KUKA KRL program: MyProgram_061().src

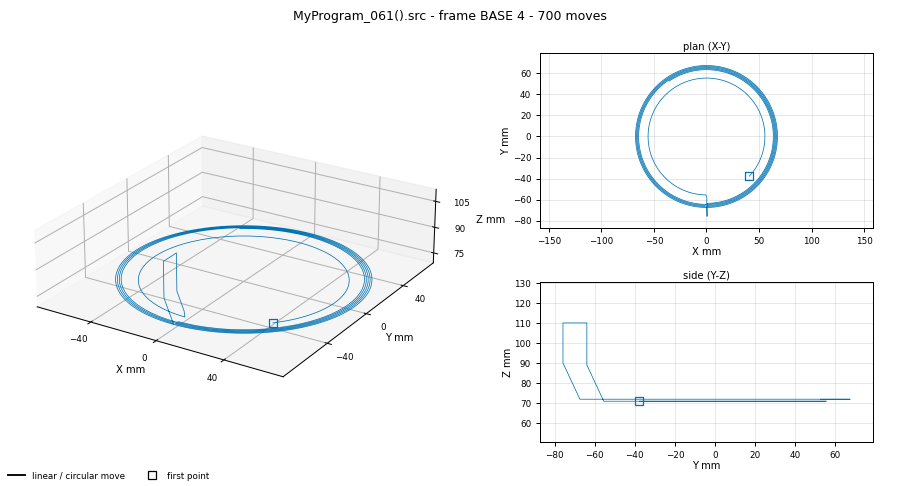
[picture p0: tool path of MyProgram_061().src in frame BASE 4, 700 of 700 moves have a stored position in this frame; points joined in program order, loops and branches not executed]
&ACCESS RVP
&REL 1
&PARAM TEMPLATE = C:\KRC\Roboter\Template\vorgabe
&PARAM EDITMASK = *
DEF MyProgram_061()
; ---- Setting reference (Base) ----
$BASE = BASE_DATA[4]

; --------------------------
; ---- Setting tool (TCP) ----
$TOOL = TOOL_DATA[3]
; --------------------------

$VEL.CP = VEL_APROX_PRINT
Startdeposition()
$VEL.CP = VEL_PRINT
LIN {X 40.7855,Y -37.7306,Z 71,A -48.0847,B 24.8792,C -2.5364,E1 25.1188,E2 491.8257} C_DIS
LIN {X 42.5102,Y -35.7771,Z 71,A -45.3429,B 24.8785,C -2.5444,E1 25.1238,E2 489.0774} C_DIS
LIN {X 44.2041,Y -33.6616,Z 71,A -42.6319,B 24.8779,C -2.5499,E1 25.1284,E2 486.3663} C_DIS
LIN {X 45.8213,Y -31.4249,Z 71,A -39.8032,B 24.8772,C -2.5572,E1 25.133,E2 483.534} C_DIS
LIN {X 47.3036,Y -29.1458,Z 71,A -37.0157,B 24.8765,C -2.5647,E1 25.1372,E2 480.7429} C_DIS
LIN {X 48.6728,Y -26.7969,Z 71,A -34.2291,B 24.8758,C -2.5723,E1 25.141,E2 477.9528} C_DIS
LIN {X 49.9338,Y -24.3666,Z 71,A -31.4273,B 24.875,C -2.58,E1 25.1445,E2 475.1476} C_DIS
LIN {X 51.0618,Y -21.9043,Z 71,A -28.6512,B 24.8743,C -2.588,E1 25.1477,E2 472.3679} C_DIS
LIN {X 52.067,Y -19.3938,Z 71,A -25.8775,B 24.8735,C -2.5961,E1 25.1505,E2 469.5904} C_DIS
LIN {X 52.9977,Y -16.6824,Z 71,A -22.8688,B 24.8725,C -2.6063,E1 25.1531,E2 466.5745} C_DIS
LIN {X 53.7819,Y -13.9471,Z 71,A -20.1757,B 24.8721,C -2.61,E1 25.1551,E2 463.8883} C_DIS
LIN {X 54.3576,Y -11.5051,Z 71,A -17.4095,B 24.8709,C -2.6221,E1 25.1568,E2 461.1095} C_DIS
LIN {X 54.8557,Y -8.8296,Z 71,A -14.6731,B 24.8702,C -2.6293,E1 25.1581,E2 458.372} C_DIS
LIN {X 55.2222,Y -6.1331,Z 71,A -11.877,B 24.8693,C -2.638,E1 25.159,E2 455.572} C_DIS
LIN {X 55.4575,Y -3.4024,Z 71,A -9.0827,B 24.8685,C -2.6462,E1 25.1596,E2 452.7749} C_DIS
LIN {X 55.5576,Y -0.6863,Z 71,A -6.4218,B 24.868,C -2.6518,E1 25.1598,E2 450.1164} C_DIS
LIN {X 55.5389,Y 1.5638,Z 71,A -3.9956,B 24.867,C -2.6615,E1 25.1596,E2 447.6817} C_DIS
LIN {X 55.3961,Y 4.2773,Z 71,A -1.3374,B 24.8664,C -2.6671,E1 25.1592,E2 445.0262} C_DIS
LIN {X 55.1439,Y 6.8016,Z 71,A 1.3866,B 24.8654,C -2.6776,E1 25.1583,E2 442.2934} C_DIS
LIN {X 54.7385,Y 9.5288,Z 71,A 4.1852,B 24.8646,C -2.6854,E1 25.1571,E2 439.4928} C_DIS
LIN {X 54.2118,Y 12.1736,Z 71,A 6.9784,B 24.8637,C -2.6941,E1 25.1555,E2 436.6953} C_DIS
LIN {X 53.5481,Y 14.8228,Z 71,A 9.7696,B 24.8629,C -2.702,E1 25.1535,E2 433.9015} C_DIS
LIN {X 52.7577,Y 17.428,Z 71,A 12.5599,B 24.8621,C -2.7099,E1 25.1511,E2 431.1084} C_DIS
LIN {X 51.8407,Y 19.9914,Z 71,A 15.3543,B 24.8613,C -2.7177,E1 25.1484,E2 428.3112} C_DIS
LIN {X 50.7941,Y 22.5183,Z 71,A 18.1681,B 24.8605,C -2.7255,E1 25.1453,E2 425.4943} C_DIS
LIN {X 49.6211,Y 24.997,Z 71,A 20.959,B 24.8598,C -2.7324,E1 25.1419,E2 422.7019} C_DIS
LIN {X 48.3402,Y 27.3922,Z 71,A 23.7438,B 24.859,C -2.7395,E1 25.1381,E2 419.9148} C_DIS
LIN {X 46.9433,Y 29.7227,Z 71,A 26.5321,B 24.8583,C -2.7464,E1 25.134,E2 417.1244} C_DIS
LIN {X 45.4343,Y 31.9818,Z 71,A 29.3209,B 24.8576,C -2.7531,E1 25.1296,E2 414.3334} C_DIS
LIN {X 43.7975,Y 34.1891,Z 71,A 32.1302,B 24.857,C -2.7593,E1 25.1248,E2 411.5228} C_DIS
LIN {X 42.0906,Y 36.2695,Z 71,A 34.9435,B 24.8562,C -2.7665,E1 25.1198,E2 408.7054} C_DIS
LIN {X 40.2294,Y 38.3236,Z 71,A 37.7223,B 24.8558,C -2.771,E1 25.1145,E2 405.9281} C_DIS
LIN {X 38.2353,Y 40.3127,Z 71,A 40.5586,B 24.8553,C -2.7755,E1 25.1088,E2 403.0929} C_DIS
LIN {X 36.2958,Y 42.0682,Z 71,A 43.3203,B 24.8546,C -2.7821,E1 25.103,E2 400.3266} C_DIS
LIN {X 34.1743,Y 43.809,Z 71,A 46.1312,B 24.8541,C -2.7868,E1 25.0969,E2 397.5151} C_DIS
LIN {X 32.0025,Y 45.4197,Z 71,A 48.9143,B 24.8536,C -2.7914,E1 25.0906,E2 394.7309} C_DIS
LIN {X 29.7582,Y 46.9206,Z 71,A 51.7458,B 24.8531,C -2.7967,E1 25.084,E2 391.8961} C_DIS
LIN {X 27.3868,Y 48.3433,Z 71,A 54.5334,B 24.8528,C -2.7994,E1 25.0773,E2 389.1106} C_DIS
LIN {X 24.9889,Y 49.6252,Z 71,A 57.3299,B 24.8524,C -2.8028,E1 25.0703,E2 386.3137} C_DIS
LIN {X 22.5309,Y 50.7884,Z 71,A 60.127,B 24.8521,C -2.8059,E1 25.0632,E2 383.5165} C_DIS
LIN {X 19.9947,Y 51.8394,Z 71,A 62.9475,B 24.8518,C -2.8085,E1 25.0559,E2 380.6962} C_DIS
LIN {X 17.4667,Y 52.7447,Z 71,A 65.7093,B 24.8516,C -2.8106,E1 25.0486,E2 377.9346} C_DIS
LIN {X 14.9277,Y 53.5184,Z 71,A 68.4748,B 24.8513,C -2.8131,E1 25.0412,E2 375.168} C_DIS
LIN {X 12.592,Y 54.1151,Z 71,A 70.7615,B 24.8516,C -2.8106,E1 25.035,E2 372.8907} C_DIS
LIN {X 10.1591,Y 54.6251,Z 71,A 73.4917,B 24.8511,C -2.8149,E1 25.0275,E2 370.1534} C_DIS
LIN {X 7.4737,Y 55.0568,Z 71,A 76.2953,B 24.8511,C -2.8156,E1 25.0198,E2 367.3507} C_DIS
LIN {X 4.7701,Y 55.3567,Z 71,A 79.1017,B 24.8511,C -2.816,E1 25.012,E2 364.5452} C_DIS
LIN {X 2.0552,Y 55.5237,Z 71,A 81.9069,B 24.8511,C -2.8159,E1 25.0042,E2 361.7412} C_DIS
LIN {X -0.664,Y 55.5577,Z 71,A 84.7191,B 24.8511,C -2.8155,E1 24.9963,E2 358.93} C_DIS
LIN {X -3.4053,Y 55.4574,Z 71,A 87.5443,B 24.8512,C -2.8144,E1 24.9884,E2 356.1067} C_DIS
LIN {X -6.1165,Y 55.2241,Z 71,A 90.3538,B 24.8513,C -2.8131,E1 24.9806,E2 353.2988} C_DIS
LIN {X -8.8133,Y 54.8583,Z 71,A 93.1693,B 24.8515,C -2.8114,E1 24.9729,E2 350.4849} C_DIS
LIN {X -11.5059,Y 54.3574,Z 71,A 96.0147,B 24.8517,C -2.8095,E1 24.9651,E2 347.6407} C_DIS
LIN {X -14.1791,Y 53.722,Z 71,A 98.8304,B 24.852,C -2.8065,E1 24.9575,E2 344.8282} C_DIS
LIN {X -16.7864,Y 52.9653,Z 71,A 101.6378,B 24.8524,C -2.8035,E1 24.95,E2 342.023} C_DIS
LIN {X -19.3546,Y 52.0818,Z 71,A 104.4495,B 24.8527,C -2.8003,E1 24.9426,E2 339.2136} C_DIS
LIN {X -21.8759,Y 51.074,Z 71,A 107.2582,B 24.8531,C -2.7965,E1 24.9353,E2 336.4075} C_DIS
LIN {X -24.3441,Y 49.9446,Z 71,A 110.0665,B 24.8535,C -2.7924,E1 24.9283,E2 333.6018} C_DIS
LIN {X -26.7824,Y 48.6807,Z 71,A 112.9149,B 24.854,C -2.788,E1 24.9212,E2 330.7559} C_DIS
LIN {X -29.1655,Y 47.2914,Z 71,A 115.7613,B 24.8545,C -2.783,E1 24.9144,E2 327.9129} C_DIS
LIN {X -31.4351,Y 45.8143,Z 71,A 118.5701,B 24.855,C -2.7779,E1 24.9079,E2 325.1068} C_DIS
LIN {X -33.7143,Y 44.1634,Z 71,A 121.4177,B 24.8558,C -2.7711,E1 24.9016,E2 322.2654} C_DIS
LIN {X -35.7726,Y 42.514,Z 71,A 124.2222,B 24.8562,C -2.7667,E1 24.8955,E2 319.4609} C_DIS
LIN {X -37.8107,Y 40.7119,Z 71,A 127.0522,B 24.8568,C -2.7607,E1 24.8897,E2 316.6336} C_DIS
LIN {X -39.8347,Y 38.7332,Z 71,A 129.9652,B 24.8576,C -2.7537,E1 24.8839,E2 313.725} C_DIS
LIN {X -41.6587,Y 36.7646,Z 71,A 132.8235,B 24.8581,C -2.7484,E1 24.8786,E2 310.8667} C_DIS
LIN {X -43.4432,Y 34.6373,Z 71,A 135.5659,B 24.8591,C -2.7391,E1 24.8737,E2 308.1339} C_DIS
LIN {X -45.0343,Y 32.5426,Z 71,A 138.3662,B 24.8597,C -2.7333,E1 24.8691,E2 305.3339} C_DIS
LIN {X -46.5685,Y 30.3066,Z 71,A 141.1834,B 24.8604,C -2.726,E1 24.8647,E2 302.52} C_DIS
LIN {X -47.9924,Y 27.997,Z 71,A 144.0124,B 24.8612,C -2.7187,E1 24.8607,E2 299.6939} C_DIS
LIN {X -49.3328,Y 25.561,Z 71,A 146.8831,B 24.862,C -2.7105,E1 24.8569,E2 296.8276} C_DIS
LIN {X -50.5224,Y 23.1212,Z 71,A 149.7025,B 24.8628,C -2.7026,E1 24.8535,E2 294.0117} C_DIS
LIN {X -51.5925,Y 20.6235,Z 71,A 152.525,B 24.8636,C -2.6946,E1 24.8505,E2 291.1927} C_DIS
LIN {X -52.5394,Y 18.0757,Z 71,A 155.3492,B 24.8645,C -2.6864,E1 24.8479,E2 288.372} C_DIS
LIN {X -53.3604,Y 15.4846,Z 71,A 158.172,B 24.8653,C -2.6782,E1 24.8456,E2 285.5528} C_DIS
LIN {X -54.0535,Y 12.8577,Z 71,A 160.9937,B 24.8662,C -2.6698,E1 24.8437,E2 282.7347} C_DIS
LIN {X -54.6257,Y 10.1558,Z 71,A 163.8614,B 24.867,C -2.6612,E1 24.8421,E2 279.8705} C_DIS
LIN {X -55.0575,Y 7.469,Z 71,A 166.6885,B 24.8679,C -2.6527,E1 24.841,E2 277.0469} C_DIS
LIN {X -55.3572,Y 4.7635,Z 71,A 169.5161,B 24.8687,C -2.6442,E1 24.8402,E2 274.2227} C_DIS
LIN {X -55.5241,Y 2.0464,Z 71,A 172.3494,B 24.8696,C -2.6357,E1 24.8398,E2 271.3926} C_DIS
LIN {X -55.56,Y -0.4299,Z 71,A 174.8514,B 24.8704,C -2.6269,E1 24.8398,E2 268.8967} C_DIS
LIN {X -55.4828,Y -2.9443,Z 71,A 177.5293,B 24.8711,C -2.6201,E1 24.8401,E2 266.2188} C_DIS
LIN {X -55.2942,Y -5.4464,Z 71,A -179.8635,B 24.8719,C -2.6123,E1 24.8408,E2 263.6146} C_DIS
LIN {X -54.9612,Y -8.1474,Z 71,A -177.0114,B 24.8727,C -2.6044,E1 24.8418,E2 260.7645} C_DIS
LIN {X -54.4945,Y -10.8382,Z 71,A -174.2087,B 24.8735,C -2.5955,E1 24.8433,E2 257.9663} C_DIS
LIN {X -53.9151,Y -13.425,Z 71,A -171.4694,B 24.8743,C -2.5874,E1 24.845,E2 255.2304} C_DIS
LIN {X -53.1514,Y -16.1868,Z 71,A -168.5076,B 24.8752,C -2.5787,E1 24.8473,E2 252.2722} C_DIS
LIN {X -52.3124,Y -18.7222,Z 71,A -165.7033,B 24.8759,C -2.5715,E1 24.8499,E2 249.4691} C_DIS
LIN {X -51.3364,Y -21.2529,Z 71,A -162.8859,B 24.8766,C -2.5639,E1 24.8528,E2 246.6542} C_DIS
LIN {X -50.2388,Y -23.731,Z 71,A -160.0738,B 24.8773,C -2.5565,E1 24.8561,E2 243.8446} C_DIS
LIN {X -49.0001,Y -26.1936,Z 71,A -157.2124,B 24.878,C -2.5491,E1 24.8597,E2 240.9854} C_DIS
LIN {X -47.6589,Y -28.5612,Z 71,A -154.3882,B 24.8787,C -2.5421,E1 24.8637,E2 238.1633} C_DIS
LIN {X -46.1931,Y -30.8757,Z 71,A -151.55,B 24.8794,C -2.5352,E1 24.868,E2 235.3274} C_DIS
LIN {X -44.6291,Y -33.0961,Z 71,A -148.7308,B 24.88,C -2.5287,E1 24.8726,E2 232.5099} C_DIS
LIN {X -42.9587,Y -35.2372,Z 71,A -145.9154,B 24.8806,C -2.5224,E1 24.8776,E2 229.6963} C_DIS
LIN {X -41.1159,Y -37.3705,Z 71,A -143.3335,B 24.8817,C -2.5104,E1 24.8823,E2 227.1315} C_DIS
LIN {X -39.7683,Y -38.8021,Z 71,A -140.955,B 24.8815,C -2.5122,E1 24.8869,E2 224.7385} C_DIS
LIN {X -37.8194,Y -40.7039,Z 71,A -138.1256,B 24.882,C -2.5069,E1 24.8926,E2 221.91} C_DIS
LIN {X -35.7707,Y -42.5156,Z 71,A -135.3035,B 24.8825,C -2.5016,E1 24.8986,E2 219.0895} C_DIS
LIN {X -33.6515,Y -44.2118,Z 71,A -132.4917,B 24.883,C -2.4969,E1 24.9048,E2 216.2787} C_DIS
LIN {X -31.4296,Y -45.818,Z 71,A -129.6545,B 24.8834,C -2.4924,E1 24.9113,E2 213.4423} C_DIS
LIN {X -29.1493,Y -47.3015,Z 71,A -126.8378,B 24.8838,C -2.4884,E1 24.9179,E2 210.6261} C_DIS
LIN {X -26.7993,Y -48.6714,Z 71,A -124.0239,B 24.8841,C -2.4848,E1 24.9248,E2 207.8127} C_DIS
LIN {X -24.3849,Y -49.9247,Z 71,A -121.2021,B 24.8844,C -2.4817,E1 24.9318,E2 204.9908} C_DIS
LIN {X -21.9003,Y -51.0636,Z 71,A -118.3881,B 24.8847,C -2.4786,E1 24.939,E2 202.1774} C_DIS
LIN {X -19.4007,Y -52.0644,Z 71,A -115.6085,B 24.8849,C -2.4761,E1 24.9462,E2 199.3979} C_DIS
LIN {X -16.8768,Y -52.9361,Z 71,A -112.8159,B 24.8851,C -2.4747,E1 24.9536,E2 196.6035} C_DIS
LIN {X -14.1541,Y -53.7287,Z 71,A -109.9102,B 24.8853,C -2.4725,E1 24.9614,E2 193.6984} C_DIS
LIN {X -11.4997,Y -54.3587,Z 71,A -107.1003,B 24.8853,C -2.4711,E1 24.9691,E2 190.8882} C_DIS
LIN {X -8.8264,Y -54.8562,Z 71,A -104.2941,B 24.8855,C -2.4703,E1 24.9768,E2 188.0813} C_DIS
LIN {X -6.0909,Y -55.2268,Z 71,A -101.4709,B 24.8855,C -2.4694,E1 24.9846,E2 185.2583} C_DIS
LIN {X -3.424,Y -55.4561,Z 71,A -98.6835,B 24.8855,C -2.4699,E1 24.9924,E2 182.4685} C_DIS
LIN {X -0.6806,Y -55.5576,Z 71,A -95.8539,B 24.8855,C -2.4703,E1 25.0003,E2 179.6376} C_DIS
LIN {X -0.6806,Y -55.5576,Z 71,A -95.8539,B 24.8855,C -2.4703,E1 25.0003,E2 179.6376} C_DIS
Enddeposition()
LIN {X 0.3163,Y -57.6707,Z 75.5315,A -95.798,B 24.8876,C -2.4468,E1 25.0003,E2 179.6376} C_DIS
LIN {X 0.3163,Y -64.01,Z 89.1262,A -95.7703,B 24.8887,C -2.4352,E1 25.0003,E2 179.6376} C_DIS
LIN {X 0.3163,Y -64.01,Z 110.1262,A -96.1254,B 24.8746,C -2.5845,E1 25.0003,E2 179.6376} C_DIS
LIN {X 0.541,Y -75.9406,Z 110.1262,A -95.0218,B 24.8919,C -2.4005,E1 25.0022,E2 178.9714} C_DIS
LIN {X 0.541,Y -75.9406,Z 90.1262,A -94.6838,B 24.9043,C -2.2582,E1 25.0022,E2 178.9714} C_DIS
LIN {X 0.4673,Y -69.6018,Z 76.5315,A -94.7092,B 24.9034,C -2.2689,E1 25.0022,E2 178.9714} C_DIS
LIN {X 0.4427,Y -67.4888,Z 72,A -94.7192,B 24.9031,C -2.2731,E1 25.0022,E2 178.9714} C_DIS
Startdeposition()
$VEL.CP = VEL_PRINT
LIN {X 3.0465,Y -67.4239,Z 72,A -92.1859,B 24.9023,C -2.2817,E1 25.0093,E2 176.4184} C_DIS
LIN {X 6.0645,Y -67.2198,Z 72,A -89.6068,B 24.9022,C -2.2832,E1 25.0165,E2 173.837} C_DIS
LIN {X 9.1586,Y -66.8693,Z 72,A -86.9568,B 24.902,C -2.285,E1 25.0238,E2 171.1848} C_DIS
LIN {X 12.2813,Y -66.3668,Z 72,A -84.2475,B 24.9018,C -2.2877,E1 25.0313,E2 168.4721} C_DIS
LIN {X 15.4225,Y -65.7074,Z 72,A -81.5243,B 24.9016,C -2.2901,E1 25.0387,E2 165.7467} C_DIS
LIN {X 18.5712,Y -64.8876,Z 72,A -78.7625,B 24.9014,C -2.293,E1 25.0462,E2 162.9825} C_DIS
LIN {X 21.7049,Y -63.9076,Z 72,A -76.0971,B 24.9014,C -2.2933,E1 25.0532,E2 160.3215} C_DIS
LIN {X 24.2902,Y -62.9701,Z 72,A -73.6943,B 24.9009,C -2.2981,E1 25.0595,E2 157.9123} C_DIS
LIN {X 27.1714,Y -61.7821,Z 72,A -71.1416,B 24.9008,C -2.2996,E1 25.0661,E2 155.3622} C_DIS
LIN {X 29.6034,Y -60.654,Z 72,A -68.807,B 24.9003,C -2.3047,E1 25.072,E2 153.0217} C_DIS
LIN {X 32.339,Y -59.2409,Z 72,A -66.2034,B 24.9,C -2.3088,E1 25.0784,E2 150.4157} C_DIS
LIN {X 34.9059,Y -57.7657,Z 72,A -63.7033,B 24.8996,C -2.313,E1 25.0844,E2 147.9133} C_DIS
LIN {X 37.4976,Y -56.1191,Z 72,A -61.0796,B 24.8991,C -2.3184,E1 25.0906,E2 145.2853} C_DIS
LIN {X 39.9919,Y -54.3685,Z 72,A -58.5313,B 24.8988,C -2.3227,E1 25.0964,E2 142.7359} C_DIS
LIN {X 42.3805,Y -52.5279,Z 72,A -55.9926,B 24.8983,C -2.3276,E1 25.1019,E2 140.195} C_DIS
LIN {X 44.7089,Y -50.562,Z 72,A -53.3854,B 24.8978,C -2.3339,E1 25.1074,E2 137.583} C_DIS
LIN {X 46.945,Y -48.4917,Z 72,A -50.8158,B 24.8973,C -2.3395,E1 25.1127,E2 135.0108} C_DIS
LIN {X 49.0787,Y -46.331,Z 72,A -48.2593,B 24.8968,C -2.3453,E1 25.1176,E2 132.4517} C_DIS
LIN {X 51.126,Y -44.063,Z 72,A -45.6236,B 24.8961,C -2.3529,E1 25.1225,E2 129.8098} C_DIS
LIN {X 53.0915,Y -41.6726,Z 72,A -43.0659,B 24.8957,C -2.3579,E1 25.127,E2 127.2522} C_DIS
LIN {X 54.915,Y -39.2379,Z 72,A -40.4951,B 24.8951,C -2.3646,E1 25.1312,E2 124.678} C_DIS
LIN {X 56.5978,Y -36.7707,Z 72,A -37.9346,B 24.8944,C -2.3722,E1 25.1352,E2 122.1121} C_DIS
LIN {X 58.206,Y -34.1668,Z 72,A -35.4034,B 24.8939,C -2.3778,E1 25.1388,E2 119.5808} C_DIS
LIN {X 59.6481,Y -31.5816,Z 72,A -32.9259,B 24.8933,C -2.3841,E1 25.1421,E2 117.1014} C_DIS
LIN {X 61.0128,Y -28.8569,Z 72,A -30.3627,B 24.8927,C -2.3911,E1 25.1453,E2 114.5355} C_DIS
LIN {X 62.1377,Y -26.3475,Z 72,A -27.976,B 24.892,C -2.3995,E1 25.1479,E2 112.1419} C_DIS
LIN {X 63.2638,Y -23.5158,Z 72,A -25.3796,B 24.8912,C -2.4076,E1 25.1505,E2 109.5408} C_DIS
LIN {X 64.2794,Y -20.5783,Z 72,A -22.9172,B 24.8909,C -2.4109,E1 25.1527,E2 107.0845} C_DIS
LIN {X 65.1078,Y -17.784,Z 72,A -20.3281,B 24.8899,C -2.4217,E1 25.1547,E2 104.4847} C_DIS
LIN {X 65.8872,Y -14.6361,Z 72,A -17.6072,B 24.8892,C -2.4295,E1 25.1564,E2 101.7613} C_DIS
LIN {X 66.5071,Y -11.4985,Z 72,A -14.9145,B 24.8885,C -2.4374,E1 25.1578,E2 99.0655} C_DIS
LIN {X 66.9708,Y -8.382,Z 72,A -12.2544,B 24.8878,C -2.4455,E1 25.1588,E2 96.402} C_DIS
LIN {X 67.2899,Y -5.2298,Z 72,A -9.6286,B 24.8871,C -2.4523,E1 25.1594,E2 93.7757} C_DIS
LIN {X 67.4554,Y -2.2519,Z 72,A -7.2372,B 24.8867,C -2.4565,E1 25.1597,E2 91.3886} C_DIS
LIN {X 67.4915,Y 0.4178,Z 72,A -4.8546,B 24.8858,C -2.4668,E1 25.1597,E2 88.9957} C_DIS
LIN {X 67.4063,Y 3.4277,Z 72,A -2.3161,B 24.8851,C -2.4744,E1 25.1595,E2 86.4544} C_DIS
LIN {X 67.1879,Y 6.4104,Z 72,A 0.2495,B 24.8843,C -2.4831,E1 25.1589,E2 83.8835} C_DIS
LIN {X 66.8007,Y 9.6406,Z 72,A 2.962,B 24.8836,C -2.4903,E1 25.1579,E2 81.1698} C_DIS
LIN {X 66.2999,Y 12.6333,Z 72,A 5.5603,B 24.8828,C -2.4989,E1 25.1566,E2 78.5667} C_DIS
LIN {X 65.6663,Y 15.5947,Z 72,A 8.0256,B 24.8823,C -2.5038,E1 25.1551,E2 76.1039} C_DIS
LIN {X 64.8876,Y 18.5712,Z 72,A 10.7132,B 24.8814,C -2.5137,E1 25.1531,E2 73.4084} C_DIS
LIN {X 63.9076,Y 21.7049,Z 72,A 13.4393,B 24.8808,C -2.5203,E1 25.1507,E2 70.6823} C_DIS
LIN {X 62.8914,Y 24.4943,Z 72,A 15.9577,B 24.8801,C -2.5275,E1 25.1482,E2 68.1608} C_DIS
LIN {X 61.7026,Y 27.3509,Z 72,A 18.5237,B 24.8795,C -2.5333,E1 25.1454,E2 65.5952} C_DIS
LIN {X 60.5094,Y 29.8978,Z 72,A 20.9549,B 24.8788,C -2.541,E1 25.1424,E2 63.1587} C_DIS
LIN {X 59.1291,Y 32.5443,Z 72,A 23.4386,B 24.8783,C -2.5465,E1 25.1392,E2 60.6751} C_DIS
LIN {X 57.6425,Y 35.1086,Z 72,A 25.9449,B 24.8777,C -2.5528,E1 25.1356,E2 58.1666} C_DIS
LIN {X 56.0135,Y 37.6538,Z 72,A 28.4811,B 24.8771,C -2.5586,E1 25.1317,E2 55.6296} C_DIS
LIN {X 54.1976,Y 40.2238,Z 72,A 31.1214,B 24.8766,C -2.5643,E1 25.1274,E2 52.9886} C_DIS
LIN {X 52.3853,Y 42.5564,Z 72,A 33.6271,B 24.876,C -2.5701,E1 25.123,E2 50.4808} C_DIS
LIN {X 50.4214,Y 44.8663,Z 72,A 36.1653,B 24.8755,C -2.575,E1 25.1184,E2 47.9425} C_DIS
LIN {X 48.339,Y 47.1035,Z 72,A 38.8042,B 24.8749,C -2.5817,E1 25.1133,E2 45.2991} C_DIS
LIN {X 46.1557,Y 49.2436,Z 72,A 41.3855,B 24.8744,C -2.5867,E1 25.1081,E2 42.7168} C_DIS
LIN {X 43.88,Y 51.2819,Z 72,A 43.9525,B 24.874,C -2.591,E1 25.1027,E2 40.1497} C_DIS
LIN {X 41.5192,Y 53.2126,Z 72,A 46.5487,B 24.8735,C -2.5958,E1 25.097,E2 37.5516} C_DIS
LIN {X 39.0793,Y 55.0281,Z 72,A 49.0988,B 24.8731,C -2.5994,E1 25.0912,E2 35.002} C_DIS
LIN {X 36.5704,Y 56.7265,Z 72,A 51.6334,B 24.8728,C -2.6025,E1 25.0853,E2 32.4685} C_DIS
LIN {X 33.9857,Y 58.3128,Z 72,A 54.2359,B 24.8724,C -2.607,E1 25.0791,E2 29.8635} C_DIS
LIN {X 31.4163,Y 59.7351,Z 72,A 56.6926,B 24.8722,C -2.6094,E1 25.0731,E2 27.4082} C_DIS
LIN {X 28.7113,Y 61.0818,Z 72,A 59.2802,B 24.8718,C -2.613,E1 25.0665,E2 24.8188} C_DIS
LIN {X 25.9706,Y 62.2965,Z 72,A 61.8519,B 24.8715,C -2.6164,E1 25.0599,E2 22.2451} C_DIS
LIN {X 23.2826,Y 63.3499,Z 72,A 64.2289,B 24.8715,C -2.6169,E1 25.0537,E2 19.8722} C_DIS
LIN {X 20.5783,Y 64.2794,Z 72,A 66.7005,B 24.8711,C -2.6199,E1 25.0472,E2 17.3981} C_DIS
LIN {X 17.7452,Y 65.1183,Z 72,A 69.2101,B 24.871,C -2.6216,E1 25.0404,E2 14.8886} C_DIS
LIN {X 14.6361,Y 65.8872,Z 72,A 71.9324,B 24.8708,C -2.6231,E1 25.033,E2 12.1665} C_DIS
LIN {X 11.4985,Y 66.5071,Z 72,A 74.6419,B 24.8708,C -2.624,E1 25.0256,E2 9.4579} C_DIS
LIN {X 8.382,Y 66.9708,Z 72,A 77.3195,B 24.8706,C -2.6247,E1 25.0182,E2 6.7809} C_DIS
LIN {X 5.2298,Y 67.2899,Z 72,A 79.9634,B 24.8707,C -2.6239,E1 25.0109,E2 4.1405} C_DIS
LIN {X 2.2519,Y 67.4554,Z 72,A 82.4866,B 24.8707,C -2.6236,E1 25.0038,E2 1.6189} C_DIS
LIN {X -0.7474,Y 67.4894,Z 72,A 85.0764,B 24.8707,C -2.6241,E1 24.9966,E2 -0.9719} C_DIS
LIN {X -3.8737,Y 67.3816,Z 72,A 87.6859,B 24.8709,C -2.6221,E1 24.9893,E2 -3.5774} C_DIS
LIN {X -6.8348,Y 67.146,Z 72,A 90.2461,B 24.8709,C -2.6218,E1 24.9822,E2 -6.1381} C_DIS
LIN {X -9.937,Y 66.7583,Z 72,A 92.9278,B 24.871,C -2.6208,E1 24.9748,E2 -8.8195} C_DIS
LIN {X -13.0653,Y 66.2168,Z 72,A 95.6433,B 24.8712,C -2.6192,E1 24.9673,E2 -11.534} C_DIS
LIN {X -16.2094,Y 65.5177,Z 72,A 98.3879,B 24.8714,C -2.6169,E1 24.9599,E2 -14.277} C_DIS
LIN {X -19.3582,Y 64.6572,Z 72,A 101.1678,B 24.8717,C -2.6142,E1 24.9524,E2 -17.0549} C_DIS
LIN {X -22.1483,Y 63.7555,Z 72,A 103.6299,B 24.872,C -2.6106,E1 24.9459,E2 -19.513} C_DIS
LIN {X -25.1936,Y 62.6149,Z 72,A 106.3976,B 24.8724,C -2.6071,E1 24.9387,E2 -22.2784} C_DIS
LIN {X -27.9427,Y 61.4372,Z 72,A 108.8432,B 24.873,C -2.6013,E1 24.9325,E2 -24.716} C_DIS
LIN {X -30.3456,Y 60.2863,Z 72,A 111.2055,B 24.873,C -2.6,E1 24.9266,E2 -27.0813} C_DIS
LIN {X -33.0501,Y 58.8471,Z 72,A 113.8218,B 24.8735,C -2.596,E1 24.9202,E2 -29.6954} C_DIS
LIN {X -35.6777,Y 57.292,Z 72,A 116.3871,B 24.874,C -2.5907,E1 24.914,E2 -32.2561} C_DIS
LIN {X -38.1834,Y 55.6547,Z 72,A 118.9897,B 24.8743,C -2.5871,E1 24.908,E2 -34.8589} C_DIS
LIN {X -40.6561,Y 53.8736,Z 72,A 121.5739,B 24.8749,C -2.5818,E1 24.9022,E2 -37.4396} C_DIS
LIN {X -43.0289,Y 51.998,Z 72,A 124.148,B 24.8754,C -2.5765,E1 24.8966,E2 -40.0106} C_DIS
LIN {X -45.3374,Y 49.9994,Z 72,A 126.8218,B 24.8758,C -2.5724,E1 24.891,E2 -42.6852} C_DIS
LIN {X -47.5542,Y 47.8946,Z 72,A 129.3811,B 24.8764,C -2.5656,E1 24.8859,E2 -45.2389} C_DIS
LIN {X -49.6741,Y 45.692,Z 72,A 131.9761,B 24.877,C -2.5592,E1 24.881,E2 -47.8301} C_DIS
LIN {X -51.691,Y 43.3985,Z 72,A 134.6032,B 24.8776,C -2.5534,E1 24.8762,E2 -50.4553} C_DIS
LIN {X -53.5973,Y 41.02,Z 72,A 137.2147,B 24.8782,C -2.5471,E1 24.8717,E2 -53.0642} C_DIS
LIN {X -55.4146,Y 38.529,Z 72,A 139.8081,B 24.8789,C -2.5396,E1 24.8675,E2 -55.6523} C_DIS
LIN {X -57.0869,Y 36.0061,Z 72,A 142.4013,B 24.8796,C -2.533,E1 24.8636,E2 -58.2428} C_DIS
LIN {X -58.6142,Y 33.4615,Z 72,A 144.947,B 24.8802,C -2.5264,E1 24.86,E2 -60.786} C_DIS
LIN {X -59.9534,Y 30.9994,Z 72,A 147.374,B 24.8807,C -2.5205,E1 24.8569,E2 -63.2117} C_DIS
LIN {X -61.2512,Y 28.3471,Z 72,A 149.751,B 24.8817,C -2.5105,E1 24.854,E2 -65.5776} C_DIS
LIN {X -62.3553,Y 25.8284,Z 72,A 152.1685,B 24.8822,C -2.5052,E1 24.8514,E2 -67.9959} C_DIS
LIN {X -63.3499,Y 23.2826,Z 72,A 154.5101,B 24.8828,C -2.4986,E1 24.8491,E2 -70.335} C_DIS
LIN {X -64.2794,Y 20.5783,Z 72,A 156.9047,B 24.8836,C -2.4905,E1 24.847,E2 -72.7239} C_DIS
LIN {X -65.1078,Y 17.784,Z 72,A 159.5197,B 24.884,C -2.4858,E1 24.845,E2 -75.3427} C_DIS
LIN {X -65.8872,Y 14.6361,Z 72,A 162.2791,B 24.8848,C -2.4773,E1 24.8432,E2 -78.098} C_DIS
LIN {X -66.5071,Y 11.4985,Z 72,A 165.0103,B 24.8856,C -2.4691,E1 24.8418,E2 -80.8258} C_DIS
LIN {X -66.9708,Y 8.382,Z 72,A 167.7085,B 24.8863,C -2.4611,E1 24.8408,E2 -83.521} C_DIS
LIN {X -67.2899,Y 5.2298,Z 72,A 170.3719,B 24.8872,C -2.4521,E1 24.8401,E2 -86.1788} C_DIS
LIN {X -67.4554,Y 2.2519,Z 72,A 172.9057,B 24.8879,C -2.4441,E1 24.8398,E2 -88.7088} C_DIS
LIN {X -67.4883,Y -0.8282,Z 72,A 175.6393,B 24.8884,C -2.4383,E1 24.8398,E2 -91.4449} C_DIS
LIN {X -67.3666,Y -4.1388,Z 72,A 178.4361,B 24.8893,C -2.4291,E1 24.8402,E2 -94.2367} C_DIS
LIN {X -67.1014,Y -7.2607,Z 72,A -178.9165,B 24.89,C -2.4205,E1 24.8409,E2 -96.8795} C_DIS
LIN {X -66.7041,Y -10.2871,Z 72,A -176.2767,B 24.8907,C -2.4135,E1 24.842,E2 -99.5183} C_DIS
LIN {X -66.1961,Y -13.1672,Z 72,A -173.8198,B 24.8914,C -2.4053,E1 24.8432,E2 -101.9702} C_DIS
LIN {X -65.5177,Y -16.2094,Z 72,A -171.0941,B 24.892,C -2.399,E1 24.845,E2 -104.6967} C_DIS
LIN {X -64.6572,Y -19.3582,Z 72,A -168.3022,B 24.8927,C -2.3912,E1 24.8471,E2 -107.4861} C_DIS
LIN {X -63.7555,Y -22.1483,Z 72,A -165.8304,B 24.8934,C -2.3835,E1 24.8493,E2 -109.9537} C_DIS
LIN {X -62.6149,Y -25.1936,Z 72,A -163.053,B 24.8941,C -2.3759,E1 24.8521,E2 -112.7286} C_DIS
LIN {X -61.4372,Y -27.9427,Z 72,A -160.5998,B 24.8949,C -2.367,E1 24.8549,E2 -115.174} C_DIS
LIN {X -60.2863,Y -30.3456,Z 72,A -158.2315,B 24.8952,C -2.3631,E1 24.8578,E2 -117.5457} C_DIS
LIN {X -58.8471,Y -33.0501,Z 72,A -155.6093,B 24.8958,C -2.3566,E1 24.8613,E2 -120.1662} C_DIS
LIN {X -57.292,Y -35.6777,Z 72,A -153.0395,B 24.8964,C -2.3494,E1 24.865,E2 -122.732} C_DIS
LIN {X -55.6547,Y -38.1834,Z 72,A -150.4334,B 24.8969,C -2.3444,E1 24.8691,E2 -125.3392} C_DIS
LIN {X -53.8736,Y -40.6561,Z 72,A -147.8471,B 24.8974,C -2.3382,E1 24.8734,E2 -127.9231} C_DIS
LIN {X -51.998,Y -43.0289,Z 72,A -145.272,B 24.8979,C -2.3324,E1 24.8779,E2 -130.4964} C_DIS
LIN {X -49.9994,Y -45.3374,Z 72,A -142.5983,B 24.8983,C -2.3284,E1 24.8829,E2 -133.1725} C_DIS
LIN {X -47.8946,Y -47.5542,Z 72,A -140.0405,B 24.8988,C -2.3221,E1 24.8878,E2 -135.7264} C_DIS
LIN {X -45.692,Y -49.6741,Z 72,A -137.448,B 24.8993,C -2.3168,E1 24.8931,E2 -138.3169} C_DIS
LIN {X -43.3985,Y -51.691,Z 72,A -134.8246,B 24.8997,C -2.3126,E1 24.8987,E2 -140.9404} C_DIS
LIN {X -41.02,Y -53.5973,Z 72,A -132.2312,B 24.9,C -2.3082,E1 24.9044,E2 -143.5328} C_DIS
LIN {X -38.529,Y -55.4146,Z 72,A -129.6413,B 24.9005,C -2.3032,E1 24.9103,E2 -146.1198} C_DIS
LIN {X -36.0061,Y -57.0869,Z 72,A -127.0448,B 24.9008,C -2.2999,E1 24.9163,E2 -148.7168} C_DIS
LIN {X -33.4615,Y -58.6142,Z 72,A -124.5074,B 24.901,C -2.2968,E1 24.9225,E2 -151.2544} C_DIS
LIN {X -30.8472,Y -60.0311,Z 72,A -121.994,B 24.9013,C -2.2933,E1 24.9287,E2 -153.7665} C_DIS
LIN {X -28.1059,Y -61.3621,Z 72,A -119.4231,B 24.9016,C -2.29,E1 24.9352,E2 -156.336} C_DIS
LIN {X -25.3076,Y -62.5685,Z 72,A -116.8629,B 24.9019,C -2.2867,E1 24.9417,E2 -158.8944} C_DIS
LIN {X -22.7376,Y -63.5472,Z 72,A -114.4786,B 24.9019,C -2.2858,E1 24.948,E2 -161.2813} C_DIS
LIN {X -19.7118,Y -64.5507,Z 72,A -111.6974,B 24.9019,C -2.2856,E1 24.9554,E2 -164.0669} C_DIS
LIN {X -16.5631,Y -65.4293,Z 72,A -108.9395,B 24.9022,C -2.2835,E1 24.9629,E2 -166.824} C_DIS
LIN {X -13.498,Y -66.1292,Z 72,A -106.4449,B 24.9026,C -2.2782,E1 24.9696,E2 -169.3091} C_DIS
LIN {X -10.717,Y -66.6377,Z 72,A -103.8593,B 24.9023,C -2.2819,E1 24.9768,E2 -171.9059} C_DIS
LIN {X -7.6073,Y -67.0631,Z 72,A -101.2066,B 24.9023,C -2.2811,E1 24.9841,E2 -174.5588} C_DIS
LIN {X -4.5313,Y -67.3404,Z 72,A -98.6084,B 24.9024,C -2.2805,E1 24.9914,E2 -177.1566} C_DIS
LIN {X -1.4981,Y -67.4766,Z 72,A -96.0673,B 24.9024,C -2.28,E1 24.9985,E2 -179.6968} C_DIS
LIN {X 0.4427,Y -67.4888,Z 72,A -94.7197,B 24.9031,C -2.2731,E1 25.0022,E2 -181.028} C_DIS
Enddeposition()
LIN {X 0.4427,Y -67.4888,Z 72,A -94.7197,B 24.9031,C -2.2731,E1 25.0022,E2 -181.028} C_DIS
Startdeposition()
$VEL.CP = VEL_PRINT
LIN {X -1.8903,Y -66.4875,Z 72,A -97.6111,B 24.9034,C -2.2687,E1 24.9941,E2 -178.1261} C_DIS
LIN {X -3.7975,Y -66.4058,Z 72,A -99.9353,B 24.9048,C -2.2529,E1 24.9875,E2 -175.7636} C_DIS
LIN {X -7.7565,Y -66.0604,Z 72,A -102.9874,B 24.904,C -2.2618,E1 24.9791,E2 -172.7307} C_DIS
LIN {X -11.7555,Y -65.4671,Z 72,A -106.308,B 24.9036,C -2.2665,E1 24.9699,E2 -169.4182} C_DIS
LIN {X -15.8202,Y -64.6054,Z 72,A -109.6264,B 24.903,C -2.2741,E1 24.9609,E2 -166.1137} C_DIS
LIN {X -18.6166,Y -63.8557,Z 72,A -112.2626,B 24.9031,C -2.2724,E1 24.9538,E2 -163.4694} C_DIS
LIN {X -21.2756,Y -63.0197,Z 72,A -114.7255,B 24.9031,C -2.2729,E1 24.9473,E2 -161.0031} C_DIS
LIN {X -24.2246,Y -61.9461,Z 72,A -117.4313,B 24.9029,C -2.2753,E1 24.9402,E2 -158.2973} C_DIS
LIN {X -27.0816,Y -60.7516,Z 72,A -119.9264,B 24.9023,C -2.2818,E1 24.9338,E2 -155.8122} C_DIS
LIN {X -30.7111,Y -58.9998,Z 72,A -123.5232,B 24.9022,C -2.2833,E1 24.9248,E2 -152.2093} C_DIS
LIN {X -32.6542,Y -57.9474,Z 72,A -125.5379,B 24.9022,C -2.2833,E1 24.9199,E2 -150.189} C_DIS
LIN {X -37.2856,Y -55.081,Z 72,A -129.9977,B 24.9011,C -2.2955,E1 24.9094,E2 -145.7437} C_DIS
LIN {X -39.5289,Y -53.4947,Z 72,A -132.5761,B 24.9011,C -2.2948,E1 24.9035,E2 -143.1549} C_DIS
LIN {X -41.9352,Y -51.6292,Z 72,A -135.2225,B 24.9008,C -2.2991,E1 24.8977,E2 -140.5087} C_DIS
LIN {X -43.9835,Y -49.8967,Z 72,A -137.5438,B 24.9005,C -2.3032,E1 24.8928,E2 -138.1883} C_DIS
LIN {X -46.2784,Y -47.7752,Z 72,A -140.2075,B 24.8999,C -2.3092,E1 24.8874,E2 -135.5279} C_DIS
LIN {X -48.3697,Y -45.6565,Z 72,A -142.7819,B 24.8995,C -2.3145,E1 24.8825,E2 -132.9549} C_DIS
LIN {X -50.3965,Y -43.4103,Z 72,A -145.4369,B 24.8991,C -2.3192,E1 24.8776,E2 -130.2994} C_DIS
LIN {X -52.0563,Y -41.4043,Z 72,A -147.7442,B 24.8987,C -2.3231,E1 24.8735,E2 -127.9905} C_DIS
LIN {X -53.4647,Y -39.5696,Z 72,A -149.7304,B 24.8983,C -2.328,E1 24.8702,E2 -126.0065} C_DIS
LIN {X -55.2907,Y -36.9759,Z 72,A -152.4302,B 24.8977,C -2.3355,E1 24.8659,E2 -123.3112} C_DIS
LIN {X -56.6684,Y -34.8269,Z 72,A -154.7142,B 24.8973,C -2.3394,E1 24.8625,E2 -121.0248} C_DIS
LIN {X -58.2658,Y -32.0833,Z 72,A -157.3909,B 24.8966,C -2.3478,E1 24.8589,E2 -118.3542} C_DIS
LIN {X -59.6257,Y -29.4773,Z 72,A -159.6069,B 24.8954,C -2.3611,E1 24.8561,E2 -116.1582} C_DIS
LIN {X -60.6778,Y -27.2461,Z 72,A -162.2325,B 24.8958,C -2.3569,E1 24.853,E2 -113.5081} C_DIS
LIN {X -62.2864,Y -23.3364,Z 72,A -165.8387,B 24.8948,C -2.368,E1 24.8493,E2 -109.9083} C_DIS
LIN {X -63.6264,Y -19.3876,Z 72,A -169.3816,B 24.8937,C -2.3795,E1 24.8462,E2 -106.3727} C_DIS
LIN {X -64.4748,Y -16.3456,Z 72,A -172.1163,B 24.893,C -2.3874,E1 24.8443,E2 -103.6409} C_DIS
LIN {X -65.2819,Y -12.745,Z 72,A -175.3901,B 24.8923,C -2.3952,E1 24.8424,E2 -100.3665} C_DIS
LIN {X -65.8217,Y -9.5741,Z 72,A -178.1276,B 24.8915,C -2.4044,E1 24.8412,E2 -97.6347} C_DIS
LIN {X -66.2133,Y -6.3226,Z 72,A 179.0603,B 24.8907,C -2.4134,E1 24.8403,E2 -94.8272} C_DIS
LIN {X -66.4237,Y -3.4727,Z 72,A 176.7966,B 24.8896,C -2.4251,E1 24.8399,E2 -92.5777} C_DIS
LIN {X -66.511,Y -0.7311,Z 72,A 174.172,B 24.8894,C -2.4273,E1 24.8398,E2 -89.9427} C_DIS
LIN {X -66.4712,Y 2.3989,Z 72,A 171.499,B 24.8886,C -2.4363,E1 24.84,E2 -87.2751} C_DIS
LIN {X -66.2997,Y 5.3376,Z 72,A 168.9504,B 24.8879,C -2.4441,E1 24.8405,E2 -84.7297} C_DIS
LIN {X -66.0058,Y 8.2117,Z 72,A 166.4414,B 24.8872,C -2.4516,E1 24.8412,E2 -82.2237} C_DIS
LIN {X -65.5841,Y 11.0848,Z 72,A 164.0005,B 24.8864,C -2.4607,E1 24.8423,E2 -79.7899} C_DIS
LIN {X -65.174,Y 13.2846,Z 72,A 161.9952,B 24.8859,C -2.4652,E1 24.8434,E2 -77.7836} C_DIS
LIN {X -64.461,Y 16.3995,Z 72,A 159.1586,B 24.8853,C -2.4721,E1 24.8452,E2 -74.9469} C_DIS
LIN {X -63.5907,Y 19.5037,Z 72,A 156.4405,B 24.8844,C -2.4819,E1 24.8474,E2 -72.2363} C_DIS
LIN {X -62.3809,Y 23.082,Z 72,A 153.1122,B 24.8836,C -2.4903,E1 24.8504,E2 -68.9093} C_DIS
LIN {X -61.2097,Y 26.0295,Z 72,A 150.3531,B 24.8829,C -2.498,E1 24.8534,E2 -66.1532} C_DIS
LIN {X -60.0078,Y 28.6918,Z 72,A 147.2526,B 24.8833,C -2.4938,E1 24.8571,E2 -63.026} C_DIS
LIN {X -57.8819,Y 32.7714,Z 72,A 143.8192,B 24.8812,C -2.5157,E1 24.8616,E2 -59.6266} C_DIS
LIN {X -56.2388,Y 35.5163,Z 72,A 141.0781,B 24.8804,C -2.5237,E1 24.8656,E2 -56.8906} C_DIS
LIN {X -54.5464,Y 38.0637,Z 72,A 138.7079,B 24.8793,C -2.5362,E1 24.8693,E2 -54.5386} C_DIS
LIN {X -53.4828,Y 39.5451,Z 72,A 136.8407,B 24.8794,C -2.5344,E1 24.8724,E2 -52.658} C_DIS
LIN {X -51.6671,Y 41.8885,Z 72,A 134.3135,B 24.8787,C -2.5416,E1 24.8768,E2 -50.1361} C_DIS
LIN {X -49.7184,Y 44.1844,Z 72,A 130.9266,B 24.8796,C -2.5321,E1 24.8831,E2 -46.7113} C_DIS
LIN {X -47.4328,Y 46.6292,Z 72,A 128.9479,B 24.8772,C -2.5574,E1 24.8868,E2 -44.7844} C_DIS
LIN {X -44.869,Y 49.1002,Z 72,A 125.5496,B 24.8772,C -2.5577,E1 24.8938,E2 -41.3728} C_DIS
LIN {X -41.9174,Y 51.6431,Z 72,A 121.8749,B 24.8772,C -2.5585,E1 24.9017,E2 -37.686} C_DIS
LIN {X -39.1013,Y 53.8078,Z 72,A 119.2755,B 24.8756,C -2.5742,E1 24.9074,E2 -35.1148} C_DIS
LIN {X -36.7655,Y 55.4298,Z 72,A 116.8045,B 24.8752,C -2.5785,E1 24.9131,E2 -32.6458} C_DIS
LIN {X -34.1636,Y 57.0708,Z 72,A 114.2829,B 24.8744,C -2.586,E1 24.9191,E2 -30.1343} C_DIS
LIN {X -31.8262,Y 58.4059,Z 72,A 111.8306,B 24.8744,C -2.5872,E1 24.9251,E2 -27.6776} C_DIS
LIN {X -29.1411,Y 59.7909,Z 72,A 109.5029,B 24.8734,C -2.5972,E1 24.9308,E2 -25.3676} C_DIS
LIN {X -26.6782,Y 60.9296,Z 72,A 106.8348,B 24.8737,C -2.5936,E1 24.9377,E2 -22.6843} C_DIS
LIN {X -23.7464,Y 62.131,Z 72,A 104.0833,B 24.8734,C -2.5968,E1 24.9448,E2 -19.9344} C_DIS
LIN {X -20.7856,Y 63.1832,Z 72,A 101.3533,B 24.8731,C -2.5995,E1 24.952,E2 -17.2058} C_DIS
LIN {X -18.7402,Y 63.8198,Z 72,A 98.9606,B 24.8741,C -2.5897,E1 24.9585,E2 -14.7856} C_DIS
LIN {X -14.3236,Y 64.9538,Z 72,A 95.6624,B 24.8724,C -2.607,E1 24.9674,E2 -11.5243} C_DIS
LIN {X -11.3101,Y 65.5464,Z 72,A 93.0852,B 24.872,C -2.6106,E1 24.9744,E2 -8.9528} C_DIS
LIN {X -7.6665,Y 66.0709,Z 72,A 90.1719,B 24.8713,C -2.6183,E1 24.9824,E2 -6.0557} C_DIS
LIN {X -4.2606,Y 66.3778,Z 72,A 86.3265,B 24.8731,C -2.5995,E1 24.9933,E2 -2.1638} C_DIS
LIN {X -0.9715,Y 66.5073,Z 72,A 82.9978,B 24.8741,C -2.5891,E1 25.0026,E2 1.1897} C_DIS
LIN {X 2.9774,Y 66.4476,Z 72,A 80.9969,B 24.871,C -2.6212,E1 25.008,E2 3.114} C_DIS
LIN {X 5.1495,Y 66.3147,Z 72,A 78.7397,B 24.8719,C -2.6123,E1 25.0143,E2 5.3912} C_DIS
LIN {X 8.131,Y 66.0156,Z 72,A 76.0927,B 24.8721,C -2.6104,E1 25.0217,E2 8.0409} C_DIS
LIN {X 11.1676,Y 65.5703,Z 72,A 73.4983,B 24.8721,C -2.6107,E1 25.0288,E2 10.632} C_DIS
LIN {X 13.9303,Y 65.0392,Z 72,A 70.9795,B 24.8724,C -2.6074,E1 25.0357,E2 13.1555} C_DIS
LIN {X 17.0502,Y 64.2921,Z 72,A 68.3043,B 24.8724,C -2.6079,E1 25.043,E2 15.8255} C_DIS
LIN {X 19.8523,Y 63.4826,Z 72,A 65.8243,B 24.8724,C -2.6069,E1 25.0496,E2 18.3037} C_DIS
LIN {X 22.6609,Y 62.5351,Z 72,A 63.2629,B 24.8726,C -2.6045,E1 25.0563,E2 20.8656} C_DIS
LIN {X 25.4852,Y 61.4383,Z 72,A 60.3696,B 24.8736,C -2.5951,E1 25.0639,E2 23.7746} C_DIS
LIN {X 28.9238,Y 59.8963,Z 72,A 57.4053,B 24.8733,C -2.5981,E1 25.0713,E2 26.7241} C_DIS
LIN {X 31.4553,Y 58.607,Z 72,A 54.0372,B 24.8757,C -2.5727,E1 25.0798,E2 30.1428} C_DIS
LIN {X 34.7572,Y 56.711,Z 72,A 51.6675,B 24.8741,C -2.59,E1 25.0853,E2 32.4643} C_DIS
LIN {X 37.2976,Y 55.0729,Z 72,A 49.0668,B 24.8745,C -2.5859,E1 25.0914,E2 35.0659} C_DIS
LIN {X 38.9885,Y 53.8897,Z 72,A 47.1602,B 24.8751,C -2.5798,E1 25.0957,E2 36.9805} C_DIS
LIN {X 41.331,Y 52.1142,Z 72,A 44.3076,B 24.8763,C -2.5673,E1 25.102,E2 39.852} C_DIS
LIN {X 45.4697,Y 48.5454,Z 72,A 40.0767,B 24.876,C -2.57,E1 25.1108,E2 44.0598} C_DIS
LIN {X 47.6735,Y 46.3839,Z 72,A 37.4194,B 24.8765,C -2.5644,E1 25.116,E2 46.7189} C_DIS
LIN {X 49.7688,Y 44.128,Z 72,A 34.4743,B 24.8778,C -2.5512,E1 25.1216,E2 49.6823} C_DIS
LIN {X 53.2549,Y 39.8505,Z 72,A 29.4479,B 24.8796,C -2.5331,E1 25.1302,E2 54.7278} C_DIS
LIN {X 55.8702,Y 36.0928,Z 72,A 26.1913,B 24.8788,C -2.5407,E1 25.1353,E2 57.9503} C_DIS
LIN {X 57.9279,Y 32.6892,Z 72,A 22.757,B 24.8797,C -2.5315,E1 25.1401,E2 61.3887} C_DIS
LIN {X 59.3338,Y 30.0603,Z 72,A 20.1959,B 24.8804,C -2.5247,E1 25.1434,E2 63.9523} C_DIS
LIN {X 60.7529,Y 27.0786,Z 72,A 17.4049,B 24.881,C -2.5181,E1 25.1467,E2 66.7436} C_DIS
LIN {X 61.6418,Y 24.9886,Z 72,A 15.3775,B 24.8817,C -2.5107,E1 25.1489,E2 68.7774} C_DIS
LIN {X 62.8224,Y 21.852,Z 72,A 12.54,B 24.8823,C -2.5036,E1 25.1516,E2 71.6159} C_DIS
LIN {X 63.7896,Y 18.842,Z 72,A 9.8774,B 24.883,C -2.4971,E1 25.1538,E2 74.2786} C_DIS
LIN {X 64.9318,Y 14.4244,Z 72,A 6.0409,B 24.8838,C -2.4877,E1 25.1563,E2 78.1152} C_DIS
LIN {X 65.7591,Y 9.995,Z 72,A 2.3633,B 24.8845,C -2.4811,E1 25.1581,E2 81.7868} C_DIS
LIN {X 66.3087,Y 5.225,Z 72,A -1.9665,B 24.8861,C -2.4631,E1 25.1594,E2 86.1336} C_DIS
LIN {X 66.5131,Y -0.3996,Z 72,A -6.4159,B 24.8866,C -2.4583,E1 25.1598,E2 90.5678} C_DIS
LIN {X 66.4457,Y -3.0147,Z 72,A -8.7614,B 24.8875,C -2.4488,E1 25.1596,E2 92.922} C_DIS
LIN {X 66.2995,Y -5.3395,Z 72,A -11.019,B 24.8887,C -2.4357,E1 25.1591,E2 95.1969} C_DIS
LIN {X 65.9905,Y -8.3327,Z 72,A -13.6308,B 24.8895,C -2.427,E1 25.1583,E2 97.8139} C_DIS
LIN {X 65.5232,Y -11.4418,Z 72,A -16.2926,B 24.8901,C -2.4197,E1 25.1571,E2 100.4774} C_DIS
LIN {X 65.1311,Y -13.4938,Z 72,A -18.2103,B 24.8909,C -2.4109,E1 25.156,E2 102.4047} C_DIS
LIN {X 64.5841,Y -15.9075,Z 72,A -20.1492,B 24.8911,C -2.4093,E1 25.1548,E2 104.3361} C_DIS
LIN {X 63.8286,Y -18.7095,Z 72,A -22.6327,B 24.8917,C -2.402,E1 25.1529,E2 106.8227} C_DIS
LIN {X 63.008,Y -21.3102,Z 72,A -24.9951,B 24.8924,C -2.3944,E1 25.1508,E2 109.1896} C_DIS
LIN {X 61.9174,Y -24.2975,Z 72,A -27.7719,B 24.8933,C -2.3851,E1 25.1481,E2 111.973} C_DIS
LIN {X 60.7099,Y -27.1749,Z 72,A -30.4435,B 24.8939,C -2.3775,E1 25.1451,E2 114.648} C_DIS
LIN {X 59.3256,Y -30.0764,Z 72,A -32.8222,B 24.8937,C -2.3796,E1 25.1422,E2 117.0088} C_DIS
LIN {X 58.2137,Y -32.177,Z 72,A -35.8618,B 24.8966,C -2.3478,E1 25.1381,E2 120.1078} C_DIS
LIN {X 56.0125,Y -35.8711,Z 72,A -38.8281,B 24.8958,C -2.3565,E1 25.1338,E2 123.0383} C_DIS
LIN {X 53.6295,Y -39.3448,Z 72,A -42.4782,B 24.8967,C -2.3461,E1 25.1279,E2 126.6952} C_DIS
LIN {X 51.7523,Y -41.7833,Z 72,A -45.1165,B 24.8973,C -2.3395,E1 25.1233,E2 129.3368} C_DIS
LIN {X 50.4799,Y -43.3125,Z 72,A -47.0555,B 24.8982,C -2.3293,E1 25.1198,E2 131.2911} C_DIS
LIN {X 47.7604,Y -46.2937,Z 72,A -50.2745,B 24.8984,C -2.3273,E1 25.1137,E2 134.5007} C_DIS
LIN {X 45.5489,Y -48.471,Z 72,A -52.9173,B 24.8989,C -2.3218,E1 25.1083,E2 137.1456} C_DIS
LIN {X 43.2816,Y -50.5061,Z 72,A -55.2331,B 24.8987,C -2.3237,E1 25.1035,E2 139.4475} C_DIS
LIN {X 41.5322,Y -51.9549,Z 72,A -57.8591,B 24.9005,C -2.3024,E1 25.0977,E2 142.114} C_DIS
LIN {X 38.3381,Y -54.3546,Z 72,A -60.9307,B 24.9003,C -2.3047,E1 25.0908,E2 145.1693} C_DIS
LIN {X 35.7619,Y -56.0826,Z 72,A -63.5771,B 24.9007,C -2.3003,E1 25.0847,E2 147.8176} C_DIS
LIN {X 32.8439,Y -57.8404,Z 72,A -67.3341,B 24.9029,C -2.2745,E1 25.0755,E2 151.6242} C_DIS
LIN {X 29.7151,Y -59.5079,Z 72,A -69.3766,B 24.9012,C -2.2946,E1 25.0705,E2 153.6136} C_DIS
LIN {X 27.2349,Y -60.6828,Z 72,A -71.9188,B 24.9019,C -2.2865,E1 25.064,E2 156.1684} C_DIS
LIN {X 24.8961,Y -61.6795,Z 72,A -74.1493,B 24.9023,C -2.2824,E1 25.0583,E2 158.4035} C_DIS
LIN {X 21.536,Y -62.9311,Z 72,A -77.1718,B 24.9025,C -2.2801,E1 25.0503,E2 161.4254} C_DIS
LIN {X 18.6187,Y -63.8551,Z 72,A -79.7924,B 24.9027,C -2.2775,E1 25.0433,E2 164.0475} C_DIS
LIN {X 15.5605,Y -64.6684,Z 72,A -82.1501,B 24.9022,C -2.2837,E1 25.037,E2 166.3869} C_DIS
LIN {X 12.916,Y -65.2486,Z 72,A -84.8184,B 24.903,C -2.2735,E1 25.0296,E2 169.076} C_DIS
LIN {X 8.4884,Y -65.9703,Z 72,A -88.6744,B 24.9032,C -2.271,E1 25.019,E2 172.9343} C_DIS
LIN {X 5.4517,Y -66.2905,Z 72,A -91.2534,B 24.9032,C -2.2708,E1 25.0118,E2 175.5121} C_DIS
LIN {X 2.4095,Y -66.4708,Z 72,A -93.9098,B 24.9034,C -2.269,E1 25.0044,E2 178.1718} C_DIS
LIN {X 0.4493,Y -66.5031,Z 72,A -95.7488,B 24.9037,C -2.2652,E1 24.9993,E2 180.0197} C_DIS
Enddeposition()
LIN {X 0.4493,Y -66.5031,Z 72,A -95.7488,B 24.9037,C -2.2652,E1 24.9993,E2 180.0197} C_DIS
Startdeposition()
$VEL.CP = VEL_PRINT
LIN {X 1.3322,Y -65.5222,Z 72,A -93.0585,B 24.8983,C -2.3276,E1 25.0072,E2 177.1816} C_DIS
LIN {X 6.4867,Y -65.2134,Z 72,A -89.0574,B 24.8992,C -2.3174,E1 25.0182,E2 173.2067} C_DIS
LIN {X 9.404,Y -64.8575,Z 72,A -86.6537,B 24.8994,C -2.3151,E1 25.0249,E2 170.8105} C_DIS
LIN {X 12.1699,Y -64.3959,Z 72,A -84.3808,B 24.8996,C -2.3127,E1 25.0311,E2 168.5458} C_DIS
LIN {X 16.6189,Y -63.3936,Z 72,A -80.1195,B 24.8987,C -2.3231,E1 25.0427,E2 164.2659} C_DIS
LIN {X 19.5765,Y -62.5435,Z 72,A -77.4453,B 24.8985,C -2.3258,E1 25.0499,E2 161.59} C_DIS
LIN {X 22.6629,Y -61.4924,Z 72,A -74.5397,B 24.8981,C -2.3308,E1 25.0575,E2 158.6785} C_DIS
LIN {X 25.7102,Y -60.282,Z 72,A -71.3425,B 24.897,C -2.3431,E1 25.0658,E2 155.4595} C_DIS
LIN {X 29.2046,Y -58.6687,Z 72,A -68.7956,B 24.8983,C -2.3279,E1 25.0722,E2 152.9552} C_DIS
LIN {X 33.1346,Y -56.5427,Z 72,A -64.9421,B 24.8979,C -2.3333,E1 25.0816,E2 149.1002} C_DIS
LIN {X 36.4297,Y -54.4787,Z 72,A -61.193,B 24.8965,C -2.3485,E1 25.0905,E2 145.3272} C_DIS
LIN {X 39.6195,Y -52.2031,Z 72,A -57.5311,B 24.8954,C -2.3616,E1 25.0988,E2 141.6474} C_DIS
LIN {X 42.2638,Y -50.0862,Z 72,A -54.7096,B 24.8951,C -2.3645,E1 25.1048,E2 138.8297} C_DIS
LIN {X 43.9423,Y -48.6217,Z 72,A -52.8171,B 24.8948,C -2.3675,E1 25.1088,E2 136.9377} C_DIS
LIN {X 46.1782,Y -46.503,Z 72,A -49.8435,B 24.8936,C -2.3811,E1 25.1148,E2 133.9442} C_DIS
LIN {X 48.6489,Y -43.9121,Z 72,A -46.8482,B 24.8932,C -2.3854,E1 25.1204,E2 130.9521} C_DIS
LIN {X 51.527,Y -40.4959,Z 72,A -43.2187,B 24.893,C -2.3883,E1 25.1268,E2 127.3325} C_DIS
LIN {X 53.297,Y -38.1361,Z 72,A -40.0696,B 24.891,C -2.4102,E1 25.132,E2 124.1468} C_DIS
LIN {X 55.1144,Y -35.4588,Z 72,A -36.7324,B 24.889,C -2.4315,E1 25.1371,E2 120.7759} C_DIS
LIN {X 57.2135,Y -31.9612,Z 72,A -34.3717,B 24.891,C -2.4098,E1 25.1403,E2 118.4788} C_DIS
LIN {X 58.7648,Y -29.0106,Z 72,A -31.5807,B 24.8905,C -2.415,E1 25.1439,E2 115.6902} C_DIS
LIN {X 59.779,Y -26.8587,Z 72,A -29.2508,B 24.8894,C -2.4278,E1 25.1466,E2 113.3428} C_DIS
LIN {X 60.9605,Y -24.0572,Z 72,A -25.9341,B 24.887,C -2.4533,E1 25.1501,E2 109.9841} C_DIS
LIN {X 62.0736,Y -21.0189,Z 72,A -23.9463,B 24.8883,C -2.4396,E1 25.1519,E2 108.0399} C_DIS
LIN {X 62.8363,Y -18.6148,Z 72,A -21.0234,B 24.8859,C -2.4655,E1 25.1542,E2 105.0724} C_DIS
LIN {X 63.9418,Y -14.3648,Z 72,A -17.2064,B 24.8848,C -2.4769,E1 25.1567,E2 101.2506} C_DIS
LIN {X 64.8101,Y -9.7289,Z 72,A -13.7227,B 24.8852,C -2.4729,E1 25.1583,E2 97.7969} C_DIS
LIN {X 65.1935,Y -6.6887,Z 72,A -11.0251,B 24.8844,C -2.4819,E1 25.1591,E2 95.094} C_DIS
LIN {X 65.5297,Y -0.9046,Z 72,A -5.7093,B 24.8823,C -2.5045,E1 25.1598,E2 89.7562} C_DIS
LIN {X 65.3845,Y 4.4481,Z 72,A -1.3667,B 24.8817,C -2.5103,E1 25.1593,E2 85.426} C_DIS
LIN {X 65.0272,Y 8.146,Z 72,A 1.9553,B 24.8806,C -2.5224,E1 25.1583,E2 82.095} C_DIS
LIN {X 64.5033,Y 11.5857,Z 72,A 5.0381,B 24.8796,C -2.5328,E1 25.1568,E2 79.0056} C_DIS
LIN {X 63.9727,Y 14.2291,Z 72,A 7.1709,B 24.8795,C -2.5341,E1 25.1556,E2 76.8822} C_DIS
LIN {X 63.0884,Y 17.7421,Z 72,A 10.0212,B 24.8793,C -2.5353,E1 25.1536,E2 74.0454} C_DIS
LIN {X 62.4069,Y 20.0082,Z 72,A 12.4185,B 24.8779,C -2.55,E1 25.1516,E2 71.627} C_DIS
LIN {X 61.185,Y 23.4798,Z 72,A 15.6609,B 24.877,C -2.56,E1 25.1485,E2 68.3792} C_DIS
LIN {X 59.778,Y 26.8611,Z 72,A 18.4502,B 24.8771,C -2.5583,E1 25.1454,E2 65.6092} C_DIS
LIN {X 58.7951,Y 28.9488,Z 72,A 20.8222,B 24.8757,C -2.5731,E1 25.1425,E2 63.2149} C_DIS
LIN {X 55.8629,Y 34.2684,Z 72,A 26.018,B 24.8746,C -2.5841,E1 25.1354,E2 58.02} C_DIS
LIN {X 54.0352,Y 37.0844,Z 72,A 29.4355,B 24.8727,C -2.6039,E1 25.13,E2 54.5725} C_DIS
LIN {X 51.2193,Y 40.8841,Z 72,A 32.8092,B 24.8736,C -2.5943,E1 25.1244,E2 51.2377} C_DIS
LIN {X 49.626,Y 42.8045,Z 72,A 35.1364,B 24.8728,C -2.603,E1 25.1201,E2 48.9005} C_DIS
LIN {X 48.0134,Y 44.6061,Z 72,A 37.3998,B 24.872,C -2.6114,E1 25.1159,E2 46.6272} C_DIS
LIN {X 45.8025,Y 46.8736,Z 72,A 40.525,B 24.8705,C -2.6262,E1 25.1096,E2 43.4801} C_DIS
LIN {X 42.8547,Y 49.5831,Z 72,A 43.6384,B 24.8708,C -2.6233,E1 25.1032,E2 40.386} C_DIS
LIN {X 40.1934,Y 51.7635,Z 72,A 46.5547,B 24.8705,C -2.6265,E1 25.0968,E2 37.4731} C_DIS
LIN {X 37.9798,Y 53.4085,Z 72,A 48.6554,B 24.8708,C -2.6229,E1 25.0921,E2 35.3883} C_DIS
LIN {X 36.2199,Y 54.6175,Z 72,A 50.9962,B 24.8694,C -2.6376,E1 25.0866,E2 33.0206} C_DIS
LIN {X 34.1932,Y 55.9086,Z 72,A 53.2089,B 24.8688,C -2.6435,E1 25.0814,E2 30.8009} C_DIS
LIN {X 31.1758,Y 57.6454,Z 72,A 56.128,B 24.8687,C -2.6446,E1 25.0742,E2 27.8878} C_DIS
LIN {X 27.5953,Y 59.4426,Z 72,A 59.3318,B 24.869,C -2.6415,E1 25.0662,E2 24.6997} C_DIS
LIN {X 24.2066,Y 60.9012,Z 72,A 62.7259,B 24.8682,C -2.6489,E1 25.0575,E2 21.296} C_DIS
LIN {X 22.2919,Y 61.6281,Z 72,A 64.5207,B 24.8681,C -2.6506,E1 25.0528,E2 19.5008} C_DIS
LIN {X 19.3206,Y 62.623,Z 72,A 67.2612,B 24.8679,C -2.6528,E1 25.0455,E2 16.7603} C_DIS
LIN {X 16.4003,Y 63.4504,Z 72,A 70.4998,B 24.8663,C -2.6683,E1 25.0367,E2 13.4899} C_DIS
LIN {X 11.7368,Y 64.4762,Z 72,A 73.6057,B 24.8686,C -2.645,E1 25.0283,E2 10.4432} C_DIS
LIN {X 9.6312,Y 64.825,Z 72,A 75.9254,B 24.8675,C -2.6561,E1 25.0219,E2 8.0994} C_DIS
LIN {X 6.7273,Y 65.1895,Z 72,A 78.5104,B 24.8675,C -2.6572,E1 25.0147,E2 5.5138} C_DIS
LIN {X 2.285,Y 65.496,Z 72,A 82.8477,B 24.8664,C -2.6673,E1 25.0025,E2 1.1539} C_DIS
LIN {X -1.7188,Y 65.5131,Z 72,A 86.1841,B 24.8669,C -2.6627,E1 24.9932,E2 -2.1718} C_DIS
LIN {X -6.3612,Y 65.226,Z 72,A 89.8289,B 24.868,C -2.6514,E1 24.9832,E2 -5.7912} C_DIS
LIN {X -8.8273,Y 64.9387,Z 72,A 92.1877,B 24.8677,C -2.6543,E1 24.9766,E2 -8.1586} C_DIS
LIN {X -11.3455,Y 64.5464,Z 72,A 94.2682,B 24.8682,C -2.6494,E1 24.9709,E2 -10.2294} C_DIS
LIN {X -14.2264,Y 63.9733,Z 72,A 96.9321,B 24.8682,C -2.6494,E1 24.9636,E2 -12.8964} C_DIS
LIN {X -19.4961,Y 62.5686,Z 72,A 101.2515,B 24.8697,C -2.6347,E1 24.9521,E2 -17.1875} C_DIS
LIN {X -21.9445,Y 61.7523,Z 72,A 103.9799,B 24.8689,C -2.6422,E1 24.9448,E2 -19.9389} C_DIS
LIN {X -24.8963,Y 60.6228,Z 72,A 107.6213,B 24.8674,C -2.6575,E1 24.9353,E2 -23.625} C_DIS
LIN {X -28.225,Y 59.1463,Z 72,A 109.9361,B 24.8697,C -2.6339,E1 24.9295,E2 -25.8893} C_DIS
LIN {X -30.3785,Y 58.0693,Z 72,A 111.9635,B 24.8702,C -2.6288,E1 24.9245,E2 -27.9101} C_DIS
LIN {X -32.8523,Y 56.7071,Z 72,A 114.5518,B 24.8704,C -2.6271,E1 24.9182,E2 -30.5019} C_DIS
LIN {X -35.5371,Y 55.0641,Z 72,A 117.2764,B 24.871,C -2.6214,E1 24.9118,E2 -33.2216} C_DIS
LIN {X -38.4185,Y 53.0944,Z 72,A 120.3382,B 24.8715,C -2.6156,E1 24.9048,E2 -36.28} C_DIS
LIN {X -41.4505,Y 50.7611,Z 72,A 123.7117,B 24.8722,C -2.6092,E1 24.8974,E2 -39.6506} C_DIS
LIN {X -43.997,Y 48.5717,Z 72,A 126.88,B 24.8724,C -2.6074,E1 24.8908,E2 -42.8272} C_DIS
LIN {X -46.3534,Y 46.3296,Z 72,A 129.4671,B 24.8735,C -2.5954,E1 24.8856,E2 -45.3966} C_DIS
LIN {X -48.7237,Y 43.8286,Z 72,A 132.5794,B 24.8741,C -2.5901,E1 24.8797,E2 -48.5098} C_DIS
LIN {X -50.7114,Y 41.513,Z 72,A 135.2339,B 24.8747,C -2.583,E1 24.875,E2 -51.1596} C_DIS
LIN {X -52.843,Y 38.7626,Z 72,A 138.4411,B 24.8752,C -2.5783,E1 24.8696,E2 -54.371} C_DIS
LIN {X -54.5845,Y 36.2698,Z 72,A 140.9848,B 24.8761,C -2.5687,E1 24.8656,E2 -56.9044} C_DIS
LIN {X -56.2216,Y 33.6771,Z 72,A 143.6665,B 24.8768,C -2.5613,E1 24.8617,E2 -59.582} C_DIS
LIN {X -58.1838,Y 30.1591,Z 72,A 147.0442,B 24.8781,C -2.5483,E1 24.8572,E2 -62.9465} C_DIS
LIN {X -59.1303,Y 28.2585,Z 72,A 149.2431,B 24.878,C -2.5497,E1 24.8545,E2 -65.1607} C_DIS
LIN {X -60.7632,Y 24.5515,Z 72,A 152.2687,B 24.88,C -2.5288,E1 24.8512,E2 -68.1532} C_DIS
LIN {X -62.2444,Y 20.5078,Z 72,A 156.3663,B 24.8804,C -2.5239,E1 24.8474,E2 -72.2623} C_DIS
LIN {X -63.0351,Y 17.9305,Z 72,A 158.7923,B 24.881,C -2.518,E1 24.8454,E2 -74.6882} C_DIS
LIN {X -63.8378,Y 14.8209,Z 72,A 161.5668,B 24.8819,C -2.5086,E1 24.8436,E2 -77.4564} C_DIS
LIN {X -64.448,Y 11.8939,Z 72,A 164.2162,B 24.8826,C -2.5011,E1 24.8421,E2 -80.1035} C_DIS
LIN {X -64.9964,Y 8.3893,Z 72,A 167.7289,B 24.8827,C -2.4995,E1 24.8408,E2 -83.6334} C_DIS
LIN {X -65.2983,Y 5.5805,Z 72,A 169.8947,B 24.884,C -2.4856,E1 24.8402,E2 -85.779} C_DIS
LIN {X -65.4801,Y 2.6993,Z 72,A 172.4728,B 24.8847,C -2.4787,E1 24.8398,E2 -88.3561} C_DIS
LIN {X -65.5341,Y -0.4698,Z 72,A 175.3356,B 24.8853,C -2.4718,E1 24.8398,E2 -91.2196} C_DIS
LIN {X -65.4343,Y -3.6423,Z 72,A 177.7317,B 24.8868,C -2.4555,E1 24.8401,E2 -93.5912} C_DIS
LIN {X -65.2696,Y -5.9006,Z 72,A -179.9763,B 24.8868,C -2.4555,E1 24.8406,E2 -95.8971} C_DIS
LIN {X -64.9178,Y -8.9806,Z 72,A -177.2633,B 24.8876,C -2.4472,E1 24.8416,E2 -98.6062} C_DIS
LIN {X -64.3165,Y -12.5833,Z 72,A -172.9618,B 24.8864,C -2.4598,E1 24.8438,E2 -102.9633} C_DIS
LIN {X -63.4022,Y -16.5861,Z 72,A -170.8421,B 24.8902,C -2.4192,E1 24.8452,E2 -104.9985} C_DIS
LIN {X -62.869,Y -18.5048,Z 72,A -167.8973,B 24.8884,C -2.4384,E1 24.8476,E2 -108.0061} C_DIS
LIN {X -61.834,Y -21.7129,Z 72,A -165.9457,B 24.891,C -2.4096,E1 24.8493,E2 -109.9} C_DIS
LIN {X -60.0602,Y -26.2239,Z 72,A -161.7324,B 24.8922,C -2.3969,E1 24.8537,E2 -114.1067} C_DIS
LIN {X -59.308,Y -27.8823,Z 72,A -160.0031,B 24.8923,C -2.3953,E1 24.8557,E2 -115.8415} C_DIS
LIN {X -58.095,Y -30.3294,Z 72,A -157.4659,B 24.8926,C -2.3918,E1 24.8589,E2 -118.3841} C_DIS
LIN {X -56.6203,Y -33.003,Z 72,A -154.3585,B 24.8925,C -2.3938,E1 24.8632,E2 -121.5123} C_DIS
LIN {X -54.9408,Y -35.7287,Z 72,A -151.9106,B 24.8938,C -2.3794,E1 24.8669,E2 -123.9382} C_DIS
LIN {X -52.718,Y -38.9333,Z 72,A -148.4569,B 24.8944,C -2.372,E1 24.8725,E2 -127.391} C_DIS
LIN {X -50.3089,Y -41.9994,Z 72,A -145.3374,B 24.8957,C -2.358,E1 24.8779,E2 -130.4919} C_DIS
LIN {X -48.6115,Y -43.9537,Z 72,A -142.7562,B 24.8955,C -2.3596,E1 24.8827,E2 -133.0885} C_DIS
LIN {X -46.4465,Y -46.2353,Z 72,A -140.0115,B 24.896,C -2.3537,E1 24.888,E2 -135.8309} C_DIS
LIN {X -43.574,Y -48.9515,Z 72,A -136.5767,B 24.8967,C -2.3464,E1 24.8951,E2 -139.2622} C_DIS
LIN {X -40.8252,Y -51.2667,Z 72,A -133.7734,B 24.8978,C -2.3334,E1 24.9011,E2 -142.0451} C_DIS
LIN {X -38.9695,Y -52.6915,Z 72,A -131.1485,B 24.8971,C -2.3423,E1 24.907,E2 -144.7007} C_DIS
LIN {X -36.6863,Y -54.3051,Z 72,A -128.7295,B 24.8974,C -2.3379,E1 24.9126,E2 -147.1173} C_DIS
LIN {X -33.8614,Y -56.1103,Z 72,A -125.9114,B 24.898,C -2.3311,E1 24.9192,E2 -149.928} C_DIS
LIN {X -30.7165,Y -57.8916,Z 72,A -123.1178,B 24.8991,C -2.3188,E1 24.926,E2 -152.7006} C_DIS
LIN {X -28.4391,Y -59.0435,Z 72,A -120.5996,B 24.8988,C -2.3225,E1 24.9324,E2 -155.2341} C_DIS
LIN {X -25.9793,Y -60.1668,Z 72,A -118.3469,B 24.8992,C -2.3175,E1 24.9381,E2 -157.4801} C_DIS
LIN {X -23.4721,Y -61.188,Z 72,A -115.8508,B 24.8992,C -2.3181,E1 24.9446,E2 -159.9832} C_DIS
LIN {X -20.6909,Y -62.1842,Z 72,A -113.2155,B 24.8992,C -2.3172,E1 24.9516,E2 -162.6213} C_DIS
LIN {X -16.6258,Y -63.3918,Z 72,A -109.4492,B 24.8994,C -2.3161,E1 24.9617,E2 -166.3911} C_DIS
LIN {X -12.9042,Y -64.2521,Z 72,A -106.2082,B 24.8997,C -2.3123,E1 24.9705,E2 -169.6272} C_DIS
LIN {X -9.7671,Y -64.8042,Z 72,A -103.2559,B 24.8994,C -2.3154,E1 24.9787,E2 -172.5895} C_DIS
LIN {X -6.9579,Y -65.1654,Z 72,A -101.1032,B 24.9001,C -2.3076,E1 24.9846,E2 -174.725} C_DIS
LIN {X -4.1496,Y -65.4045,Z 72,A -98.2324,B 24.8993,C -2.3171,E1 24.9927,E2 -177.6195} C_DIS
LIN {X -1.5016,Y -65.5187,Z 72,A -95.5795,B 24.8985,C -2.3254,E1 25.0001,E2 -180.2924} C_DIS
LIN {X -1.5016,Y -65.5187,Z 72,A -95.5795,B 24.8985,C -2.3254,E1 25.0001,E2 -180.2924} C_DIS
Enddeposition()
LIN {X 0.4521,Y -64.5472,Z 72,A -95.5516,B 24.9004,C -2.3035,E1 25.0001,E2 -180.2685} C_DIS
Startdeposition()
$VEL.CP = VEL_PRINT
LIN {X -2.0738,Y -64.5238,Z 72,A -97.697,B 24.9003,C -2.3052,E1 24.9941,E2 -178.1269} C_DIS
LIN {X -5.0206,Y -64.3616,Z 72,A -100.6303,B 24.9009,C -2.2981,E1 24.9858,E2 -175.1756} C_DIS
LIN {X -8.1995,Y -64.0343,Z 72,A -103.3885,B 24.9007,C -2.3002,E1 24.9782,E2 -172.4207} C_DIS
LIN {X -11.1268,Y -63.5914,Z 72,A -106.7071,B 24.902,C -2.2858,E1 24.969,E2 -169.0646} C_DIS
LIN {X -16.3378,Y -62.4557,Z 72,A -111.9027,B 24.9026,C -2.2784,E1 24.9548,E2 -163.8442} C_DIS
LIN {X -20.3353,Y -61.2712,Z 72,A -114.5511,B 24.9004,C -2.3037,E1 24.9479,E2 -161.2512} C_DIS
LIN {X -23.2733,Y -60.2159,Z 72,A -116.8093,B 24.8993,C -2.3172,E1 24.9421,E2 -159.0206} C_DIS
LIN {X -25.2276,Y -59.4234,Z 72,A -118.7514,B 24.8993,C -2.3175,E1 24.9371,E2 -157.0749} C_DIS
LIN {X -29.2485,Y -57.5511,Z 72,A -122.8363,B 24.8991,C -2.3189,E1 24.9267,E2 -152.9828} C_DIS
LIN {X -30.994,Y -56.63,Z 72,A -124.8574,B 24.8994,C -2.3154,E1 24.9217,E2 -150.9479} C_DIS
LIN {X -33.6019,Y -55.1229,Z 72,A -128.0513,B 24.9,C -2.3084,E1 24.914,E2 -147.7275} C_DIS
LIN {X -36.4971,Y -53.2514,Z 72,A -131.088,B 24.8996,C -2.3137,E1 24.907,E2 -144.6932} C_DIS
LIN {X -39.3491,Y -51.1788,Z 72,A -134.4007,B 24.8994,C -2.3154,E1 24.8996,E2 -141.3726} C_DIS
LIN {X -42.0988,Y -48.9429,Z 72,A -136.8857,B 24.8977,C -2.3347,E1 24.8944,E2 -138.924} C_DIS
LIN {X -45.6821,Y -45.6167,Z 72,A -141.3003,B 24.8971,C -2.3419,E1 24.8854,E2 -134.5084} C_DIS
LIN {X -47.864,Y -43.3216,Z 72,A -143.8756,B 24.8961,C -2.3527,E1 24.8806,E2 -131.9477} C_DIS
LIN {X -49.3638,Y -41.6043,Z 72,A -146.3923,B 24.8966,C -2.3474,E1 24.876,E2 -129.4068} C_DIS
LIN {X -51.9102,Y -38.3802,Z 72,A -150.5318,B 24.8966,C -2.3464,E1 24.869,E2 -125.2452} C_DIS
LIN {X -53.7779,Y -35.7155,Z 72,A -152.2334,B 24.894,C -2.377,E1 24.8664,E2 -123.6081} C_DIS
LIN {X -55.8859,Y -32.3173,Z 72,A -156.2425,B 24.894,C -2.377,E1 24.8605,E2 -119.5785} C_DIS
LIN {X -57.3081,Y -29.7228,Z 72,A -158.6077,B 24.8929,C -2.3892,E1 24.8574,E2 -117.2298} C_DIS
LIN {X -58.0789,Y -28.186,Z 72,A -160.4803,B 24.8931,C -2.3866,E1 24.8551,E2 -115.3409} C_DIS
LIN {X -59.3162,Y -25.48,Z 72,A -163.3075,B 24.8928,C -2.3904,E1 24.8519,E2 -112.5073} C_DIS
LIN {X -60.5681,Y -22.3413,Z 72,A -166.3484,B 24.8921,C -2.3982,E1 24.8489,E2 -109.4679} C_DIS
LIN {X -62.0392,Y -17.8536,Z 72,A -169.8395,B 24.8897,C -2.4241,E1 24.846,E2 -106.0186} C_DIS
LIN {X -62.7658,Y -15.1016,Z 72,A -173.4482,B 24.8909,C -2.411,E1 24.8435,E2 -102.3574} C_DIS
LIN {X -63.8413,Y -9.5905,Z 72,A -177.92,B 24.8886,C -2.436,E1 24.8413,E2 -97.9189} C_DIS
LIN {X -64.226,Y -6.5324,Z 72,A 179.3376,B 24.8879,C -2.4444,E1 24.8404,E2 -95.1801} C_DIS
LIN {X -64.4223,Y -4.1715,Z 72,A 176.9853,B 24.8877,C -2.4463,E1 24.84,E2 -92.8182} C_DIS
LIN {X -64.5557,Y 0.4377,Z 72,A 173.0812,B 24.8862,C -2.4627,E1 24.8398,E2 -88.93} C_DIS
LIN {X -64.4629,Y 3.4867,Z 72,A 170.4045,B 24.8853,C -2.4719,E1 24.8401,E2 -86.259} C_DIS
LIN {X -63.9886,Y 8.5486,Z 72,A 165.1242,B 24.8853,C -2.4717,E1 24.8418,E2 -80.9467} C_DIS
LIN {X -63.1882,Y 13.2262,Z 72,A 161.8616,B 24.8824,C -2.5029,E1 24.8434,E2 -77.7392} C_DIS
LIN {X -62.8126,Y 14.9061,Z 72,A 160.0286,B 24.8825,C -2.5018,E1 24.8446,E2 -75.893} C_DIS
LIN {X -61.9425,Y 18.1871,Z 72,A 156.7943,B 24.882,C -2.5069,E1 24.847,E2 -72.6522} C_DIS
LIN {X -60.7134,Y 21.9427,Z 72,A 153.1626,B 24.8812,C -2.5153,E1 24.8503,E2 -69.0197} C_DIS
LIN {X -58.949,Y 26.3169,Z 72,A 149.1006,B 24.8798,C -2.5302,E1 24.8547,E2 -64.9708} C_DIS
LIN {X -57.7035,Y 28.9472,Z 72,A 145.7692,B 24.8805,C -2.5235,E1 24.8589,E2 -61.6055} C_DIS
LIN {X -55.9893,Y 32.1374,Z 72,A 143.4201,B 24.878,C -2.5491,E1 24.8621,E2 -59.3054} C_DIS
LIN {X -54.4225,Y 34.7251,Z 72,A 140.8107,B 24.8772,C -2.5581,E1 24.8659,E2 -56.704} C_DIS
LIN {X -52.2032,Y 37.98,Z 72,A 136.8387,B 24.8772,C -2.5583,E1 24.8723,E2 -52.7131} C_DIS
LIN {X -49.8677,Y 40.9991,Z 72,A 133.7889,B 24.8756,C -2.5737,E1 24.8776,E2 -49.6855} C_DIS
LIN {X -47.7269,Y 43.472,Z 72,A 131.0764,B 24.8746,C -2.5846,E1 24.8826,E2 -46.9872} C_DIS
LIN {X -45.6688,Y 45.6302,Z 72,A 128.0043,B 24.8748,C -2.5826,E1 24.8886,E2 -43.897} C_DIS
LIN {X -43.1013,Y 48.0614,Z 72,A 125.076,B 24.8737,C -2.594,E1 24.8946,E2 -40.9839} C_DIS
LIN {X -40.9106,Y 49.9395,Z 72,A 122.3042,B 24.8735,C -2.5953,E1 24.9005,E2 -38.2048} C_DIS
LIN {X -37.7353,Y 52.3806,Z 72,A 118.3587,B 24.8735,C -2.5948,E1 24.9094,E2 -34.244} C_DIS
LIN {X -34.1011,Y 54.8156,Z 72,A 115.1278,B 24.8716,C -2.6152,E1 24.9169,E2 -31.0514} C_DIS
LIN {X -31.6903,Y 56.2441,Z 72,A 112.558,B 24.8713,C -2.6179,E1 24.9231,E2 -28.4802} C_DIS
LIN {X -30.0194,Y 57.1528,Z 72,A 110.5063,B 24.8718,C -2.6132,E1 24.9282,E2 -26.4118} C_DIS
LIN {X -26.4393,Y 58.8947,Z 72,A 107.1194,B 24.871,C -2.6216,E1 24.9368,E2 -23.0364} C_DIS
LIN {X -23.1025,Y 60.2817,Z 72,A 103.1948,B 24.872,C -2.6111,E1 24.9471,E2 -19.0784} C_DIS
LIN {X -19.7246,Y 61.4702,Z 72,A 100.9796,B 24.8696,C -2.6348,E1 24.9528,E2 -16.9155} C_DIS
LIN {X -15.3903,Y 62.6958,Z 72,A 96.8675,B 24.8695,C -2.6365,E1 24.9639,E2 -12.801} C_DIS
LIN {X -12.5129,Y 63.3334,Z 72,A 94.1468,B 24.8695,C -2.6365,E1 24.9713,E2 -10.077} C_DIS
LIN {X -10.021,Y 63.7745,Z 72,A 91.7168,B 24.8697,C -2.6341,E1 24.978,E2 -7.6391} C_DIS
LIN {X -6.7073,Y 64.2077,Z 72,A 89.2265,B 24.8685,C -2.646,E1 24.9849,E2 -5.1755} C_DIS
LIN {X -3.7934,Y 64.4459,Z 72,A 86.2754,B 24.8692,C -2.6393,E1 24.9931,E2 -2.2074} C_DIS
LIN {X 0.2217,Y 64.5569,Z 72,A 82.9863,B 24.8685,C -2.6462,E1 25.0023,E2 1.0655} C_DIS
LIN {X 5.3524,Y 64.3351,Z 72,A 78.275,B 24.8688,C -2.6429,E1 25.0154,E2 5.7828} C_DIS
LIN {X 8.4091,Y 64.007,Z 72,A 75.6303,B 24.8688,C -2.6443,E1 25.0227,E2 8.4222} C_DIS
LIN {X 10.8456,Y 63.6398,Z 72,A 73.0305,B 24.8697,C -2.6344,E1 25.03,E2 11.043} C_DIS
LIN {X 17.3515,Y 62.182,Z 72,A 67.4626,B 24.8692,C -2.6391,E1 25.045,E2 16.5918} C_DIS
LIN {X 20.3654,Y 61.2613,Z 72,A 64.1574,B 24.8706,C -2.6253,E1 25.0539,E2 19.9236} C_DIS
LIN {X 26.4918,Y 58.871,Z 72,A 58.8619,B 24.8699,C -2.6319,E1 25.0675,E2 25.1913} C_DIS
LIN {X 29.4885,Y 57.4286,Z 72,A 55.8902,B 24.8703,C -2.6278,E1 25.0749,E2 28.1647} C_DIS
LIN {X 31.9859,Y 56.076,Z 72,A 53.2759,B 24.8709,C -2.6221,E1 25.0813,E2 30.7846} C_DIS
LIN {X 35.921,Y 53.6414,Z 72,A 49.3886,B 24.871,C -2.6211,E1 25.0905,E2 34.6619} C_DIS
LIN {X 37.6999,Y 52.4056,Z 72,A 47.0768,B 24.8722,C -2.6086,E1 25.0958,E2 36.9953} C_DIS
LIN {X 42.029,Y 49.0023,Z 72,A 42.8891,B 24.8715,C -2.6165,E1 25.1048,E2 41.1484} C_DIS
LIN {X 44.9991,Y 46.2901,Z 72,A 38.9856,B 24.873,C -2.6012,E1 25.1128,E2 45.0722} C_DIS
LIN {X 46.9956,Y 44.2609,Z 72,A 36.5152,B 24.8734,C -2.5972,E1 25.1176,E2 47.5416} C_DIS
LIN {X 49.8423,Y 41.0299,Z 72,A 32.465,B 24.8747,C -2.5829,E1 25.125,E2 51.6071} C_DIS
LIN {X 53.0453,Y 36.7942,Z 72,A 27.5701,B 24.8763,C -2.567,E1 25.1331,E2 56.5161} C_DIS
LIN {X 55.0348,Y 33.7469,Z 72,A 24.1251,B 24.8776,C -2.5534,E1 25.1382,E2 59.9759} C_DIS
LIN {X 58.0362,Y 28.2743,Z 72,A 19.6061,B 24.8766,C -2.564,E1 25.144,E2 64.446} C_DIS
LIN {X 59.3029,Y 25.5102,Z 72,A 16.3322,B 24.8787,C -2.5419,E1 25.1478,E2 67.7543} C_DIS
LIN {X 60.5222,Y 22.4633,Z 72,A 13.4844,B 24.8794,C -2.5352,E1 25.1506,E2 70.6022} C_DIS
LIN {X 61.6421,Y 19.1801,Z 72,A 10.7854,B 24.8793,C -2.5357,E1 25.153,E2 73.2846} C_DIS
LIN {X 62.4011,Y 16.5423,Z 72,A 7.7651,B 24.8814,C -2.5136,E1 25.1552,E2 76.3398} C_DIS
LIN {X 63.2929,Y 12.7132,Z 72,A 4.8024,B 24.8811,C -2.5164,E1 25.157,E2 79.2787} C_DIS
LIN {X 63.745,Y 10.2117,Z 72,A 2.5307,B 24.8818,C -2.509,E1 25.158,E2 81.5546} C_DIS
LIN {X 64.1318,Y 7.398,Z 72,A -0.1623,B 24.883,C -2.4968,E1 25.159,E2 84.2606} C_DIS
LIN {X 64.4012,Y 4.4856,Z 72,A -2.3634,B 24.8828,C -2.4987,E1 25.1595,E2 86.444} C_DIS
LIN {X 64.5348,Y 1.6944,Z 72,A -5.3968,B 24.8849,C -2.4767,E1 25.1598,E2 89.5113} C_DIS
LIN {X 64.5495,Y -0.9985,Z 72,A -7.9571,B 24.886,C -2.4648,E1 25.1597,E2 92.0845} C_DIS
LIN {X 64.1913,Y -6.8635,Z 72,A -12.9881,B 24.8871,C -2.453,E1 25.1585,E2 97.1136} C_DIS
LIN {X 63.5853,Y -11.1611,Z 72,A -16.2805,B 24.8869,C -2.4552,E1 25.1571,E2 100.3815} C_DIS
LIN {X 63.1444,Y -13.431,Z 72,A -18.2923,B 24.8874,C -2.4497,E1 25.156,E2 102.3944} C_DIS
LIN {X 62.6758,Y -15.4724,Z 72,A -20.4988,B 24.8887,C -2.435,E1 25.1546,E2 104.6229} C_DIS
LIN {X 61.4921,Y -19.6563,Z 72,A -23.7088,B 24.8883,C -2.4397,E1 25.1521,E2 107.8034} C_DIS
LIN {X 60.0033,Y -23.8168,Z 72,A -28.083,B 24.8904,C -2.4162,E1 25.1478,E2 112.2089} C_DIS
LIN {X 58.744,Y -26.7729,Z 72,A -30.7116,B 24.8907,C -2.4133,E1 25.1449,E2 114.8298} C_DIS
LIN {X 57.1273,Y -30.0678,Z 72,A -34.2601,B 24.8922,C -2.3964,E1 25.1404,E2 118.3995} C_DIS
LIN {X 54.4299,Y -34.7135,Z 72,A -38.6635,B 24.8926,C -2.3921,E1 25.1342,E2 122.7903} C_DIS
LIN {X 52.7512,Y -37.2147,Z 72,A -41.5685,B 24.8938,C -2.379,E1 25.1295,E2 125.7122} C_DIS
LIN {X 51.1762,Y -39.3525,Z 72,A -44.2752,B 24.8951,C -2.3639,E1 25.1249,E2 128.4416} C_DIS
LIN {X 48.1795,Y -42.9694,Z 72,A -48.0346,B 24.8951,C -2.3635,E1 25.1181,E2 132.1848} C_DIS
LIN {X 44.5633,Y -46.7097,Z 72,A -53.0114,B 24.8969,C -2.3435,E1 25.1083,E2 137.1879} C_DIS
LIN {X 41.7357,Y -49.2521,Z 72,A -55.8141,B 24.8964,C -2.3501,E1 25.1024,E2 139.964} C_DIS
LIN {X 39.1372,Y -51.3411,Z 72,A -59.3051,B 24.8981,C -2.3307,E1 25.0947,E2 143.4879} C_DIS
LIN {X 36.133,Y -53.4979,Z 72,A -62.9283,B 24.8994,C -2.3159,E1 25.0863,E2 147.1338} C_DIS
LIN {X 33.3136,Y -55.2981,Z 72,A -64.9503,B 24.8978,C -2.3334,E1 25.0816,E2 149.1081} C_DIS
LIN {X 29.3365,Y -57.5064,Z 72,A -69.4626,B 24.8994,C -2.315,E1 25.0704,E2 153.651} C_DIS
LIN {X 25.1227,Y -59.4682,Z 72,A -73.2984,B 24.8994,C -2.3158,E1 25.0607,E2 157.4754} C_DIS
LIN {X 22.7172,Y -60.4282,Z 72,A -75.5903,B 24.8996,C -2.3128,E1 25.0547,E2 159.7693} C_DIS
LIN {X 19.7843,Y -61.4508,Z 72,A -78.3204,B 24.8999,C -2.3101,E1 25.0475,E2 162.5007} C_DIS
LIN {X 16.7333,Y -62.3508,Z 72,A -82.1628,B 24.9022,C -2.2833,E1 25.037,E2 166.4004} C_DIS
LIN {X 12.8423,Y -63.2668,Z 72,A -84.3249,B 24.8997,C -2.3124,E1 25.0313,E2 168.4907} C_DIS
LIN {X 9.9186,Y -63.7906,Z 72,A -87.3859,B 24.9007,C -2.3005,E1 25.0228,E2 171.5769} C_DIS
LIN {X 5.427,Y -64.3292,Z 72,A -91.0597,B 24.9002,C -2.306,E1 25.0126,E2 175.2349} C_DIS
LIN {X 3.5448,Y -64.4597,Z 72,A -93.3753,B 24.9016,C -2.2907,E1 25.006,E2 177.586} C_DIS
LIN {X 0.4521,Y -64.5472,Z 72,A -95.5504,B 24.9005,C -2.303,E1 25.0001,E2 179.7315} C_DIS
Enddeposition()
LIN {X 0.4521,Y -64.5472,Z 72,A -95.5504,B 24.9005,C -2.303,E1 25.0001,E2 179.7315} C_DIS
Startdeposition()
$VEL.CP = VEL_PRINT
LIN {X 0.8268,Y -63.5735,Z 72,A -93.9143,B 24.8964,C -2.3496,E1 25.0049,E2 177.9849} C_DIS
LIN {X 3.7418,Y -63.4688,Z 72,A -91.719,B 24.8972,C -2.3406,E1 25.011,E2 175.8117} C_DIS
LIN {X 6.5427,Y -63.241,Z 72,A -88.9358,B 24.8966,C -2.3478,E1 25.0188,E2 173.0133} C_DIS
LIN {X 9.1211,Y -62.921,Z 72,A -85.9334,B 24.8951,C -2.3648,E1 25.0272,E2 169.973} C_DIS
LIN {X 12.6945,Y -62.2983,Z 72,A -82.6394,B 24.8948,C -2.3682,E1 25.0362,E2 166.675} C_DIS
LIN {X 15.8352,Y -61.5749,Z 72,A -80.6581,B 24.8965,C -2.3491,E1 25.0414,E2 164.7419} C_DIS
LIN {X 20.0029,Y -60.3504,Z 72,A -76.5902,B 24.8957,C -2.3572,E1 25.0523,E2 160.662} C_DIS
LIN {X 22.1652,Y -59.59,Z 72,A -73.8534,B 24.8941,C -2.3761,E1 25.0596,E2 157.8863} C_DIS
LIN {X 25.7742,Y -58.12,Z 72,A -71.2626,B 24.8956,C -2.3589,E1 25.0661,E2 155.3424} C_DIS
LIN {X 29.1514,Y -56.5021,Z 72,A -67.0844,B 24.8934,C -2.3839,E1 25.0767,E2 151.1163} C_DIS
LIN {X 33.096,Y -54.2853,Z 72,A -63.4195,B 24.8936,C -2.381,E1 25.0855,E2 147.4693} C_DIS
LIN {X 35.9548,Y -52.4363,Z 72,A -60.6033,B 24.8936,C -2.3808,E1 25.092,E2 144.663} C_DIS
LIN {X 38.7703,Y -50.3893,Z 72,A -57.315,B 24.8927,C -2.391,E1 25.0994,E2 141.3623} C_DIS
LIN {X 41.6584,Y -48.0284,Z 72,A -53.5777,B 24.8912,C -2.4079,E1 25.1074,E2 137.5995} C_DIS
LIN {X 44.4446,Y -45.464,Z 72,A -50.209,B 24.8906,C -2.4148,E1 25.1142,E2 134.2286} C_DIS
LIN {X 47.5115,Y -42.2484,Z 72,A -46.556,B 24.8905,C -2.4158,E1 25.1211,E2 130.5891} C_DIS
LIN {X 50.2331,Y -38.9732,Z 72,A -43.3265,B 24.891,C -2.4104,E1 25.1267,E2 127.3873} C_DIS
LIN {X 51.5653,Y -37.1929,Z 72,A -41.0106,B 24.8898,C -2.4237,E1 25.1306,E2 125.0512} C_DIS
LIN {X 52.8429,Y -35.3549,Z 72,A -38.7926,B 24.8888,C -2.4343,E1 25.1341,E2 122.8191} C_DIS
LIN {X 55.2118,Y -31.5263,Z 72,A -34.3982,B 24.8869,C -2.4544,E1 25.1404,E2 118.3996} C_DIS
LIN {X 57.291,Y -27.5675,Z 72,A -30.3688,B 24.8858,C -2.4662,E1 25.1454,E2 114.3638} C_DIS
LIN {X 58.99,Y -23.7163,Z 72,A -26.7083,B 24.8851,C -2.4742,E1 25.1494,E2 110.7048} C_DIS
LIN {X 60.5344,Y -19.4379,Z 72,A -23.2865,B 24.8856,C -2.4693,E1 25.1525,E2 107.3138} C_DIS
LIN {X 61.3053,Y -16.8489,Z 72,A -20.5257,B 24.8841,C -2.4852,E1 25.1546,E2 104.5311} C_DIS
LIN {X 62.0298,Y -13.9476,Z 72,A -17.896,B 24.8834,C -2.492,E1 25.1563,E2 101.9007} C_DIS
LIN {X 62.6301,Y -10.9433,Z 72,A -14.5739,B 24.8813,C -2.5152,E1 25.158,E2 98.5431} C_DIS
LIN {X 63.1853,Y -7.0625,Z 72,A -11.7886,B 24.882,C -2.507,E1 25.159,E2 95.7936} C_DIS
LIN {X 63.4811,Y -3.5192,Z 72,A -8.1144,B 24.8799,C -2.5293,E1 25.1597,E2 92.0885} C_DIS
LIN {X 63.5774,Y -0.3936,Z 72,A -5.9458,B 24.8807,C -2.5215,E1 25.1597,E2 89.9513} C_DIS
LIN {X 63.5586,Y 1.5911,Z 72,A -4.0905,B 24.88,C -2.5288,E1 25.1597,E2 88.0896} C_DIS
LIN {X 63.4379,Y 4.2266,Z 72,A -1.5235,B 24.8788,C -2.5412,E1 25.1593,E2 85.5088} C_DIS
LIN {X 63.1666,Y 7.2263,Z 72,A 1.2324,B 24.8779,C -2.5507,E1 25.1585,E2 82.7465} C_DIS
LIN {X 62.7109,Y 10.4677,Z 72,A 4.0643,B 24.8773,C -2.5568,E1 25.1573,E2 79.9169} C_DIS
LIN {X 62.2511,Y 12.9243,Z 72,A 6.0747,B 24.8773,C -2.5575,E1 25.1562,E2 77.9166} C_DIS
LIN {X 61.6279,Y 15.6282,Z 72,A 9.0391,B 24.8753,C -2.577,E1 25.1542,E2 74.9235} C_DIS
LIN {X 60.6603,Y 19.041,Z 72,A 11.8333,B 24.8754,C -2.5762,E1 25.152,E2 72.147} C_DIS
LIN {X 58.9988,Y 23.6943,Z 72,A 16.2102,B 24.8743,C -2.5871,E1 25.1478,E2 67.7687} C_DIS
LIN {X 57.3016,Y 27.5454,Z 72,A 20.1393,B 24.873,C -2.6011,E1 25.1433,E2 63.8278} C_DIS
LIN {X 55.5302,Y 30.9616,Z 72,A 24.1989,B 24.8706,C -2.6254,E1 25.1378,E2 59.7322} C_DIS
LIN {X 53.5927,Y 34.2064,Z 72,A 27.6563,B 24.8696,C -2.6354,E1 25.1327,E2 56.2685} C_DIS
LIN {X 50.8586,Y 38.1527,Z 72,A 31.882,B 24.8688,C -2.6434,E1 25.1258,E2 52.0443} C_DIS
LIN {X 48.8515,Y 40.6911,Z 72,A 34.8195,B 24.8681,C -2.6506,E1 25.1205,E2 49.1032} C_DIS
LIN {X 46.2206,Y 43.6566,Z 72,A 37.7745,B 24.8688,C -2.6432,E1 25.115,E2 46.1789} C_DIS
LIN {X 44.2244,Y 45.6777,Z 72,A 40.7559,B 24.8673,C -2.6588,E1 25.109,E2 43.173} C_DIS
LIN {X 41.2984,Y 48.3392,Z 72,A 44.6422,B 24.8658,C -2.6736,E1 25.1008,E2 39.267} C_DIS
LIN {X 38.7331,Y 50.4181,Z 72,A 47.5108,B 24.8655,C -2.6762,E1 25.0944,E2 36.4026} C_DIS
LIN {X 35.4204,Y 52.7986,Z 72,A 51.1517,B 24.865,C -2.6813,E1 25.086,E2 32.7621} C_DIS
LIN {X 32.5594,Y 54.6093,Z 72,A 53.848,B 24.8654,C -2.6772,E1 25.0796,E2 30.0839} C_DIS
LIN {X 29.4221,Y 56.361,Z 72,A 56.7639,B 24.8657,C -2.6738,E1 25.0725,E2 27.1842} C_DIS
LIN {X 26.883,Y 57.6154,Z 72,A 59.3383,B 24.8654,C -2.6774,E1 25.066,E2 24.6082} C_DIS
LIN {X 23.764,Y 58.9695,Z 72,A 62.2918,B 24.8654,C -2.678,E1 25.0584,E2 21.6601} C_DIS
LIN {X 20.6239,Y 60.1399,Z 72,A 65.7995,B 24.8639,C -2.692,E1 25.0491,E2 18.1264} C_DIS
LIN {X 15.6097,Y 61.6328,Z 72,A 70.6876,B 24.8632,C -2.699,E1 25.0359,E2 13.2296} C_DIS
LIN {X 9.7748,Y 62.8227,Z 72,A 75.4773,B 24.8643,C -2.6879,E1 25.0229,E2 8.4716} C_DIS
LIN {X 6.7866,Y 63.2155,Z 72,A 78.0843,B 24.8645,C -2.6859,E1 25.0157,E2 5.8713} C_DIS
LIN {X 3.4455,Y 63.4851,Z 72,A 81.4168,B 24.8638,C -2.6929,E1 25.0063,E2 2.5236} C_DIS
LIN {X 0.1041,Y 63.5791,Z 72,A 84.5482,B 24.8636,C -2.6951,E1 24.9976,E2 -0.6126} C_DIS
LIN {X -3.5646,Y 63.4785,Z 72,A 87.4614,B 24.8646,C -2.6853,E1 24.9895,E2 -3.5033} C_DIS
LIN {X -6.5007,Y 63.2454,Z 72,A 90.2156,B 24.8645,C -2.6862,E1 24.9819,E2 -6.261} C_DIS
LIN {X -9.3833,Y 62.8823,Z 72,A 92.9691,B 24.8644,C -2.6875,E1 24.9742,E2 -9.0197} C_DIS
LIN {X -13.1258,Y 62.2092,Z 72,A 96.2358,B 24.865,C -2.6813,E1 24.9653,E2 -12.2753} C_DIS
LIN {X -15.35,Y 61.6979,Z 72,A 98.6284,B 24.8645,C -2.6866,E1 24.9588,E2 -14.6838} C_DIS
LIN {X -19.5256,Y 60.5061,Z 72,A 102.2758,B 24.8655,C -2.6766,E1 24.9491,E2 -18.3137} C_DIS
LIN {X -22.6491,Y 59.4072,Z 72,A 105.2105,B 24.8659,C -2.6718,E1 24.9414,E2 -21.2428} C_DIS
LIN {X -26.6977,Y 57.701,Z 72,A 108.9941,B 24.8669,C -2.6625,E1 24.9317,E2 -25.0131} C_DIS
LIN {X -30.5998,Y 55.7314,Z 72,A 113.081,B 24.8672,C -2.6591,E1 24.9216,E2 -29.103} C_DIS
LIN {X -33.0289,Y 54.3261,Z 72,A 115.5861,B 24.8677,C -2.6541,E1 24.9156,E2 -31.6038} C_DIS
LIN {X -35.435,Y 52.7888,Z 72,A 118.4735,B 24.8676,C -2.6556,E1 24.9088,E2 -34.5043} C_DIS
Enddeposition()
END
